SPLINE
SPL {X  -143.903, Y  +318.857, Z    +0.000, E1   +34.827, E3 +27306.081}
SPL {X  -153.845, Y  +344.850, Z    +0.000, E1   +24.318, E3 +27332.176}
SPL {X  -158.184, Y  +364.762, Z    +0.000, E1   +14.458, E3 +27341.556}
SPL {X  -159.644, Y  +378.137, Z    +0.000, E1    +6.763, E3 +27344.869}
SPL {X  -159.957, Y  +385.097, Z    +0.000, E1    +2.214, E3 +27345.786}
SPL {X  -160.000, Y  +390.467, Z    +0.000, E1    -1.886, E3 +27346.226}
SPL {X  -160.000, Y  +396.882, Z    +0.000, E1    -9.361, E3 +27346.979}
SPL {X  -160.000, Y  +403.298, Z    +0.000, E1   -17.340, E3 +27348.282}
SPL {X  -160.000, Y  +414.216, Z    +0.000, E1   -29.557, E3 +27351.832}
SPL {X  -160.000, Y  +448.199, Z    +0.000, E1   -47.246, E3 +27374.324}
SPL {X  -160.000, Y  +510.996, Z    +0.000, E1   -52.996, E3 +27446.648}
SPL {X  -160.000, Y  +527.680, Z    +0.000, E1   -53.008, E3 +27473.417}
SPL {X  -160.000, Y  +543.568, Z    +0.000, E1   -52.978, E3 +27498.957}
SPL {X  -160.000, Y  +558.178, Z    +0.000, E1   -52.971, E3 +27522.417}
SPL {X  -160.000, Y  +573.149, Z    +0.000, E1   -52.983, E3 +27546.431}
SPL {X  -160.000, Y  +589.074, Z    +0.000, E1   -52.998, E3 +27571.971}
SPL {X  -160.000, Y  +605.389, Z    +0.000, E1   -52.996, E3 +27598.171}
SPL {X  -160.000, Y  +621.194, Z    +0.000, E1   -52.986, E3 +27623.571}
SPL {X  -160.000, Y  +634.261, Z    +0.000, E1   -52.926, E3 +27644.650}
SPL {X  -160.000, Y  +645.165, Z    +0.000, E1   -52.917, E3 +27662.170}
SPL {X  -160.000, Y  +655.362, Z    +0.000, E1   -52.919, E3 +27678.521}
SPL {X  -160.000, Y  +666.642, Z    +0.000, E1   -52.938, E3 +27696.596}
SPL {X  -159.882, Y  +677.646, Z    +0.000, E1   -52.897, E3 +27714.427}
SPL {X  -159.100, Y  +688.445, Z    +0.000, E1   -52.790, E3 +27732.550}
SPL {X  -157.767, Y  +698.140, Z    +0.000, E1   -52.527, E3 +27749.561}
SPL {X  -155.944, Y  +707.296, Z    +0.000, E1   -52.232, E3 +27766.119}
SPL {X  -153.388, Y  +717.020, Z    +0.000, E1   -51.781, E3 +27784.324}
SPL {X  -150.628, Y  +725.455, Z    +0.000, E1   -51.252, E3 +27800.683}
SPL {X  -147.586, Y  +733.294, Z    +0.000, E1   -50.691, E3 +27816.259}
SPL {X  -144.002, Y  +741.239, Z    +0.000, E1   -50.009, E3 +27832.435}
SPL {X  -134.968, Y  +757.427, Z    +0.000, E1   -43.006, E3 +27917.714}
ENDSPLINE

SPLINE
SPL {X  -150.251, Y  +726.498, Z    +0.000, E1   -29.147, E3 +27992.699}
SPL {X  -158.295, Y  +694.796, Z    +0.000, E1   -14.337, E3 +28010.691}
SPL {X  -159.852, Y  +678.369, Z    +0.000, E1    -4.607, E3 +28014.636}
SPL {X  -159.994, Y  +672.856, Z    +0.000, E1    -0.741, E3 +28015.223}
SPL {X  -160.000, Y  +667.974, Z    +0.000, E1    +3.384, E3 +28015.651}
SPL {X  -160.000, Y  +657.936, Z    +0.000, E1   +15.171, E3 +28017.404}
SPL {X  -160.000, Y  +643.339, Z    +0.000, E1   +31.330, E3 +28022.395}
SPL {X  -160.000, Y  +606.884, Z    +0.000, E1   +47.933, E3 +28048.251}
SPL {X  -160.000, Y  +552.863, Z    +0.000, E1   +52.205, E3 +28114.055}
SPL {X  -160.000, Y  +541.250, Z    +0.000, E1   +52.128, E3 +28133.359}
SPL {X  -160.000, Y  +532.225, Z    +0.000, E1   +52.130, E3 +28148.267}
SPL {X  -160.000, Y  +522.908, Z    +0.000, E1   +52.129, E3 +28163.671}
SPL {X  -160.000, Y  +514.018, Z    +0.000, E1   +52.121, E3 +28178.355}
SPL {X  -160.000, Y  +502.148, Z    +0.000, E1   +52.197, E3 +28197.831}
SPL {X  -160.000, Y  +488.825, Z    +0.000, E1   +51.737, E3 +28222.876}
ENDSPLINE

SPLINE
SPL {X  -160.000, Y  +489.568, Z    +0.000, E1   +48.224, E3 +28241.900}
ENDSPLINE

SPLINE
SPL {X  -160.000, Y  +479.301, Z    +0.000, E1   +49.113, E3 +28255.778}
SPL {X  -160.000, Y  +468.407, Z    +0.000, E1   +50.011, E3 +28270.105}
SPL {X  -160.000, Y  +457.258, Z    +0.000, E1   +50.929, E3 +28284.090}
SPL {X  -160.000, Y  +444.555, Z    +0.000, E1   +51.931, E3 +28299.575}
SPL {X  -160.000, Y  +432.374, Z    +0.000, E1   +52.787, E3 +28314.199}
SPL {X  -160.000, Y  +422.570, Z    +0.000, E1   +53.120, E3 +28327.957}
SPL {X  -160.000, Y  +412.343, Z    +0.000, E1   +53.116, E3 +28344.264}
SPL {X  -160.000, Y  +402.505, Z    +0.000, E1   +53.115, E3 +28359.937}
SPL {X  -160.000, Y  +391.565, Z    +0.000, E1   +53.135, E3 +28377.344}
SPL {X  -159.782, Y  +380.451, Z    +0.000, E1   +53.086, E3 +28395.306}
SPL {X  -159.005, Y  +370.988, Z    +0.000, E1   +52.949, E3 +28411.205}
SPL {X  -157.765, Y  +362.152, Z    +0.000, E1   +52.730, E3 +28426.603}
SPL {X  -156.057, Y  +353.496, Z    +0.000, E1   +52.443, E3 +28442.142}
SPL {X  -153.530, Y  +343.760, Z    +0.000, E1   +52.025, E3 +28460.195}
SPL {X  -150.540, Y  +334.599, Z    +0.000, E1   +51.451, E3 +28477.843}
SPL {X  -147.202, Y  +326.099, Z    +0.000, E1   +50.843, E3 +28494.637}
SPL {X  -143.559, Y  +318.154, Z    +0.000, E1   +50.126, E3 +28510.784}
SPL {X  -132.920, Y  +299.736, Z    +0.000, E1   +44.141, E3 +28591.929}
ENDSPLINE

SPLINE
SPL {X  -143.903, Y  +318.857, Z    +0.000, E1   +34.827, E3 +28656.076}
SPL {X  -153.845, Y  +344.850, Z    +0.000, E1   +24.318, E3 +28682.171}
SPL {X  -158.184, Y  +364.762, Z    +0.000, E1   +14.458, E3 +28691.551}
SPL {X  -159.644, Y  +378.137, Z    +0.000, E1    +6.763, E3 +28694.864}
SPL {X  -159.957, Y  +385.097, Z    +0.000, E1    +2.214, E3 +28695.781}
SPL {X  -160.000, Y  +390.467, Z    +0.000, E1    -1.886, E3 +28696.222}
SPL {X  -160.000, Y  +396.882, Z    +0.000, E1    -9.361, E3 +28696.974}
SPL {X  -160.000, Y  +403.298, Z    +0.000, E1   -17.340, E3 +28698.277}
SPL {X  -160.000, Y  +414.216, Z    +0.000, E1   -29.557, E3 +28701.827}
SPL {X  -160.000, Y  +448.199, Z    +0.000, E1   -47.246, E3 +28724.319}
SPL {X  -160.000, Y  +510.996, Z    +0.000, E1   -52.996, E3 +28796.643}
SPL {X  -160.000, Y  +527.680, Z    +0.000, E1   -53.008, E3 +28823.412}
SPL {X  -160.000, Y  +543.568, Z    +0.000, E1   -52.978, E3 +28848.952}
SPL {X  -160.000, Y  +558.178, Z    +0.000, E1   -52.971, E3 +28872.412}
SPL {X  -160.000, Y  +573.149, Z    +0.000, E1   -52.983, E3 +28896.426}
SPL {X  -160.000, Y  +589.074, Z    +0.000, E1   -52.998, E3 +28921.966}
SPL {X  -160.000, Y  +605.389, Z    +0.000, E1   -52.996, E3 +28948.167}
SPL {X  -160.000, Y  +621.194, Z    +0.000, E1   -52.986, E3 +28973.566}
SPL {X  -160.000, Y  +634.261, Z    +0.000, E1   -52.926, E3 +28994.646}
SPL {X  -160.000, Y  +645.165, Z    +0.000, E1   -52.917, E3 +29012.165}
SPL {X  -160.000, Y  +655.362, Z    +0.000, E1   -52.919, E3 +29028.516}
SPL {X  -160.000, Y  +666.642, Z    +0.000, E1   -52.938, E3 +29046.591}
SPL {X  -159.882, Y  +677.646, Z    +0.000, E1   -52.897, E3 +29064.423}
SPL {X  -159.100, Y  +688.445, Z    +0.000, E1   -52.790, E3 +29082.545}
SPL {X  -157.767, Y  +698.140, Z    +0.000, E1   -52.527, E3 +29099.556}
SPL {X  -155.944, Y  +707.296, Z    +0.000, E1   -52.232, E3 +29116.115}
SPL {X  -153.388, Y  +717.020, Z    +0.000, E1   -51.781, E3 +29134.320}
SPL {X  -150.628, Y  +725.455, Z    +0.000, E1   -51.252, E3 +29150.678}
SPL {X  -147.586, Y  +733.294, Z    +0.000, E1   -50.691, E3 +29166.255}
SPL {X  -144.002, Y  +741.239, Z    +0.000, E1   -50.009, E3 +29182.431}
SPL {X  -134.968, Y  +757.427, Z    +0.000, E1   -43.006, E3 +29267.709}
ENDSPLINE

SPLINE
SPL {X  -150.251, Y  +726.498, Z    +0.000, E1   -29.147, E3 +29342.694}
SPL {X  -158.295, Y  +694.796, Z    +0.000, E1   -14.337, E3 +29360.687}
SPL {X  -159.852, Y  +678.369, Z    +0.000, E1    -4.607, E3 +29364.631}
SPL {X  -159.994, Y  +672.856, Z    +0.000, E1    -0.741, E3 +29365.219}
SPL {X  -160.000, Y  +667.974, Z    +0.000, E1    +3.384, E3 +29365.646}
SPL {X  -160.000, Y  +657.936, Z    +0.000, E1   +15.171, E3 +29367.399}
SPL {X  -160.000, Y  +643.339, Z    +0.000, E1   +31.330, E3 +29372.390}
SPL {X  -160.000, Y  +606.884, Z    +0.000, E1   +47.933, E3 +29398.246}
SPL {X  -160.000, Y  +552.863, Z    +0.000, E1   +52.205, E3 +29464.051}
SPL {X  -160.000, Y  +541.250, Z    +0.000, E1   +52.128, E3 +29483.354}
SPL {X  -160.000, Y  +532.225, Z    +0.000, E1   +52.130, E3 +29498.262}
SPL {X  -160.000, Y  +522.908, Z    +0.000, E1   +52.129, E3 +29513.666}
SPL {X  -160.000, Y  +514.018, Z    +0.000, E1   +52.121, E3 +29528.351}
SPL {X  -160.000, Y  +502.148, Z    +0.000, E1   +52.197, E3 +29547.827}
SPL {X  -160.000, Y  +488.825, Z    +0.000, E1   +51.737, E3 +29572.871}
ENDSPLINE

SPLINE
SPL {X  -160.000, Y  +489.568, Z    +0.000, E1   +48.224, E3 +29591.896}
ENDSPLINE

SPLINE
SPL {X  -160.000, Y  +479.301, Z    +0.000, E1   +49.113, E3 +29605.774}
SPL {X  -160.000, Y  +468.407, Z    +0.000, E1   +50.011, E3 +29620.100}
SPL {X  -160.000, Y  +457.258, Z    +0.000, E1   +50.929, E3 +29634.086}
SPL {X  -160.000, Y  +444.555, Z    +0.000, E1   +51.931, E3 +29649.570}
SPL {X  -160.000, Y  +432.374, Z    +0.000, E1   +52.787, E3 +29664.194}
SPL {X  -160.000, Y  +422.570, Z    +0.000, E1   +53.120, E3 +29677.952}
SPL {X  -160.000, Y  +412.343, Z    +0.000, E1   +53.116, E3 +29694.259}
SPL {X  -160.000, Y  +402.505, Z    +0.000, E1   +53.115, E3 +29709.932}
SPL {X  -160.000, Y  +391.565, Z    +0.000, E1   +53.135, E3 +29727.339}
SPL {X  -159.782, Y  +380.451, Z    +0.000, E1   +53.086, E3 +29745.301}
SPL {X  -159.005, Y  +370.988, Z    +0.000, E1   +52.949, E3 +29761.200}
SPL {X  -157.765, Y  +362.152, Z    +0.000, E1   +52.730, E3 +29776.599}
SPL {X  -156.057, Y  +353.496, Z    +0.000, E1   +52.443, E3 +29792.137}
SPL {X  -153.530, Y  +343.760, Z    +0.000, E1   +52.025, E3 +29810.190}
SPL {X  -150.540, Y  +334.599, Z    +0.000, E1   +51.451, E3 +29827.839}
SPL {X  -147.202, Y  +326.099, Z    +0.000, E1   +50.843, E3 +29844.632}
SPL {X  -143.559, Y  +318.154, Z    +0.000, E1   +50.126, E3 +29860.779}
SPL {X  -132.920, Y  +299.736, Z    +0.000, E1   +44.141, E3 +29941.924}
ENDSPLINE

SPLINE
SPL {X  -143.903, Y  +318.857, Z    +0.000, E1   +34.827, E3 +30006.071}
SPL {X  -153.845, Y  +344.850, Z    +0.000, E1   +24.318, E3 +30032.167}
SPL {X  -158.184, Y  +364.762, Z    +0.000, E1   +14.458, E3 +30041.546}
SPL {X  -159.644, Y  +378.137, Z    +0.000, E1    +6.763, E3 +30044.860}
SPL {X  -159.957, Y  +385.097, Z    +0.000, E1    +2.214, E3 +30045.776}
SPL {X  -160.000, Y  +390.467, Z    +0.000, E1    -1.886, E3 +30046.217}
SPL {X  -160.000, Y  +396.882, Z    +0.000, E1    -9.361, E3 +30046.970}
SPL {X  -160.000, Y  +403.298, Z    +0.000, E1   -17.340, E3 +30048.272}
SPL {X  -160.000, Y  +414.216, Z    +0.000, E1   -29.557, E3 +30051.822}
SPL {X  -160.000, Y  +448.199, Z    +0.000, E1   -47.246, E3 +30074.315}
SPL {X  -160.000, Y  +510.996, Z    +0.000, E1   -52.996, E3 +30146.639}
SPL {X  -160.000, Y  +527.680, Z    +0.000, E1   -53.008, E3 +30173.407}
SPL {X  -160.000, Y  +543.568, Z    +0.000, E1   -52.978, E3 +30198.947}
SPL {X  -160.000, Y  +558.178, Z    +0.000, E1   -52.971, E3 +30222.407}
SPL {X  -160.000, Y  +573.149, Z    +0.000, E1   -52.983, E3 +30246.421}
SPL {X  -160.000, Y  +589.074, Z    +0.000, E1   -52.998, E3 +30271.961}
SPL {X  -160.000, Y  +605.389, Z    +0.000, E1   -52.996, E3 +30298.162}
SPL {X  -160.000, Y  +621.194, Z    +0.000, E1   -52.986, E3 +30323.561}
SPL {X  -160.000, Y  +634.261, Z    +0.000, E1   -52.926, E3 +30344.641}
SPL {X  -160.000, Y  +645.165, Z    +0.000, E1   -52.917, E3 +30362.160}
SPL {X  -160.000, Y  +655.362, Z    +0.000, E1   -52.919, E3 +30378.511}
SPL {X  -160.000, Y  +666.642, Z    +0.000, E1   -52.938, E3 +30396.586}
SPL {X  -159.882, Y  +677.646, Z    +0.000, E1   -52.897, E3 +30414.418}
SPL {X  -159.100, Y  +688.445, Z    +0.000, E1   -52.790, E3 +30432.540}
SPL {X  -157.767, Y  +698.140, Z    +0.000, E1   -52.527, E3 +30449.552}
SPL {X  -155.944, Y  +707.296, Z    +0.000, E1   -52.232, E3 +30466.110}
SPL {X  -153.388, Y  +717.020, Z    +0.000, E1   -51.781, E3 +30484.315}
SPL {X  -150.628, Y  +725.455, Z    +0.000, E1   -51.252, E3 +30500.673}
SPL {X  -147.586, Y  +733.294, Z    +0.000, E1   -50.691, E3 +30516.250}
SPL {X  -144.002, Y  +741.239, Z    +0.000, E1   -50.009, E3 +30532.426}
SPL {X  -134.968, Y  +757.427, Z    +0.000, E1   -43.006, E3 +30617.704}
ENDSPLINE

SPLINE
SPL {X  -150.251, Y  +726.498, Z    +0.000, E1   -29.147, E3 +30692.690}
SPL {X  -158.295, Y  +694.796, Z    +0.000, E1   -14.337, E3 +30710.682}
SPL {X  -159.852, Y  +678.369, Z    +0.000, E1    -4.607, E3 +30714.626}
SPL {X  -159.994, Y  +672.856, Z    +0.000, E1    -0.741, E3 +30715.214}
SPL {X  -160.000, Y  +667.974, Z    +0.000, E1    +3.384, E3 +30715.642}
SPL {X  -160.000, Y  +657.936, Z    +0.000, E1   +15.171, E3 +30717.394}
SPL {X  -160.000, Y  +643.339, Z    +0.000, E1   +31.330, E3 +30722.386}
SPL {X  -160.000, Y  +606.884, Z    +0.000, E1   +47.933, E3 +30748.241}
SPL {X  -160.000, Y  +552.863, Z    +0.000, E1   +52.205, E3 +30814.046}
SPL {X  -160.000, Y  +541.250, Z    +0.000, E1   +52.128, E3 +30833.350}
SPL {X  -160.000, Y  +532.225, Z    +0.000, E1   +52.130, E3 +30848.257}
SPL {X  -160.000, Y  +522.908, Z    +0.000, E1   +52.129, E3 +30863.661}
SPL {X  -160.000, Y  +514.018, Z    +0.000, E1   +52.121, E3 +30878.346}
SPL {X  -160.000, Y  +502.148, Z    +0.000, E1   +52.197, E3 +30897.822}
SPL {X  -160.000, Y  +488.825, Z    +0.000, E1   +51.737, E3 +30922.867}
ENDSPLINE

SPLINE
SPL {X  -160.000, Y  +489.568, Z    +0.000, E1   +48.224, E3 +30941.891}
ENDSPLINE

SPLINE
SPL {X  -160.000, Y  +479.301, Z    +0.000, E1   +49.113, E3 +30955.769}
SPL {X  -160.000, Y  +468.407, Z    +0.000, E1   +50.011, E3 +30970.095}
SPL {X  -160.000, Y  +457.258, Z    +0.000, E1   +50.929, E3 +30984.081}
SPL {X  -160.000, Y  +444.555, Z    +0.000, E1   +51.931, E3 +30999.565}
SPL {X  -160.000, Y  +432.374, Z    +0.000, E1   +52.787, E3 +31014.189}
SPL {X  -160.000, Y  +422.570, Z    +0.000, E1   +53.120, E3 +31027.948}
SPL {X  -160.000, Y  +412.343, Z    +0.000, E1   +53.116, E3 +31044.254}
SPL {X  -160.000, Y  +402.505, Z    +0.000, E1   +53.115, E3 +31059.927}
SPL {X  -160.000, Y  +391.565, Z    +0.000, E1   +53.135, E3 +31077.334}
SPL {X  -159.782, Y  +380.451, Z    +0.000, E1   +53.086, E3 +31095.297}
SPL {X  -159.005, Y  +370.988, Z    +0.000, E1   +52.949, E3 +31111.195}
SPL {X  -157.765, Y  +362.152, Z    +0.000, E1   +52.730, E3 +31126.594}
SPL {X  -156.057, Y  +353.496, Z    +0.000, E1   +52.443, E3 +31142.132}
SPL {X  -153.530, Y  +343.760, Z    +0.000, E1   +52.025, E3 +31160.185}
SPL {X  -150.540, Y  +334.599, Z    +0.000, E1   +51.451, E3 +31177.834}
SPL {X  -147.202, Y  +326.099, Z    +0.000, E1   +50.843, E3 +31194.627}
SPL {X  -143.559, Y  +318.154, Z    +0.000, E1   +50.126, E3 +31210.775}
SPL {X  -132.920, Y  +299.736, Z    +0.000, E1   +44.141, E3 +31291.919}
ENDSPLINE

SPLINE
SPL {X  -143.903, Y  +318.857, Z    +0.000, E1   +34.827, E3 +31356.067}
SPL {X  -153.845, Y  +344.850, Z    +0.000, E1   +24.318, E3 +31382.162}
SPL {X  -158.184, Y  +364.762, Z    +0.000, E1   +14.458, E3 +31391.541}
SPL {X  -159.644, Y  +378.137, Z    +0.000, E1    +6.763, E3 +31394.855}
SPL {X  -159.957, Y  +385.097, Z    +0.000, E1    +2.214, E3 +31395.771}
SPL {X  -160.000, Y  +390.467, Z    +0.000, E1    -1.886, E3 +31396.212}
SPL {X  -160.000, Y  +396.882, Z    +0.000, E1    -9.361, E3 +31396.965}
SPL {X  -160.000, Y  +403.298, Z    +0.000, E1   -17.340, E3 +31398.268}
SPL {X  -160.000, Y  +414.216, Z    +0.000, E1   -29.557, E3 +31401.817}
SPL {X  -160.000, Y  +448.199, Z    +0.000, E1   -47.246, E3 +31424.310}
SPL {X  -160.000, Y  +510.996, Z    +0.000, E1   -52.996, E3 +31496.634}
SPL {X  -160.000, Y  +527.680, Z    +0.000, E1   -53.008, E3 +31523.403}
SPL {X  -160.000, Y  +543.568, Z    +0.000, E1   -52.978, E3 +31548.943}
SPL {X  -160.000, Y  +558.178, Z    +0.000, E1   -52.971, E3 +31572.402}
SPL {X  -160.000, Y  +573.149, Z    +0.000, E1   -52.983, E3 +31596.416}
SPL {X  -160.000, Y  +589.074, Z    +0.000, E1   -52.998, E3 +31621.957}
SPL {X  -160.000, Y  +605.389, Z    +0.000, E1   -52.996, E3 +31648.157}
SPL {X  -160.000, Y  +621.194, Z    +0.000, E1   -52.986, E3 +31673.557}
SPL {X  -160.000, Y  +634.261, Z    +0.000, E1   -52.926, E3 +31694.636}
SPL {X  -160.000, Y  +645.165, Z    +0.000, E1   -52.917, E3 +31712.155}
SPL {X  -160.000, Y  +655.362, Z    +0.000, E1   -52.919, E3 +31728.506}
SPL {X  -160.000, Y  +666.642, Z    +0.000, E1   -52.938, E3 +31746.582}
SPL {X  -159.882, Y  +677.646, Z    +0.000, E1   -52.897, E3 +31764.413}
SPL {X  -159.100, Y  +688.445, Z    +0.000, E1   -52.790, E3 +31782.536}
SPL {X  -157.767, Y  +698.140, Z    +0.000, E1   -52.527, E3 +31799.547}
SPL {X  -155.944, Y  +707.296, Z    +0.000, E1   -52.232, E3 +31816.105}
SPL {X  -153.388, Y  +717.020, Z    +0.000, E1   -51.781, E3 +31834.310}
SPL {X  -150.628, Y  +725.455, Z    +0.000, E1   -51.252, E3 +31850.668}
SPL {X  -147.586, Y  +733.294, Z    +0.000, E1   -50.691, E3 +31866.245}
SPL {X  -144.002, Y  +741.239, Z    +0.000, E1   -50.009, E3 +31882.421}
SPL {X  -134.968, Y  +757.427, Z    +0.000, E1   -43.006, E3 +31967.700}
ENDSPLINE

SPLINE
SPL {X  -150.251, Y  +726.498, Z    +0.000, E1   -29.147, E3 +32042.685}
SPL {X  -158.295, Y  +694.796, Z    +0.000, E1   -14.337, E3 +32060.677}
SPL {X  -159.852, Y  +678.369, Z    +0.000, E1    -4.607, E3 +32064.621}
SPL {X  -159.994, Y  +672.856, Z    +0.000, E1    -0.741, E3 +32065.209}
SPL {X  -160.000, Y  +667.974, Z    +0.000, E1    +3.384, E3 +32065.637}
SPL {X  -160.000, Y  +657.936, Z    +0.000, E1   +15.171, E3 +32067.389}
SPL {X  -160.000, Y  +643.339, Z    +0.000, E1   +31.330, E3 +32072.381}
SPL {X  -160.000, Y  +606.884, Z    +0.000, E1   +47.933, E3 +32098.236}
SPL {X  -160.000, Y  +552.863, Z    +0.000, E1   +52.205, E3 +32164.041}
SPL {X  -160.000, Y  +541.250, Z    +0.000, E1   +52.128, E3 +32183.345}
SPL {X  -160.000, Y  +532.225, Z    +0.000, E1   +52.130, E3 +32198.253}
SPL {X  -160.000, Y  +522.908, Z    +0.000, E1   +52.129, E3 +32213.656}
SPL {X  -160.000, Y  +514.018, Z    +0.000, E1   +52.121, E3 +32228.341}
SPL {X  -160.000, Y  +502.148, Z    +0.000, E1   +52.197, E3 +32247.817}
SPL {X  -160.000, Y  +488.825, Z    +0.000, E1   +51.737, E3 +32272.862}
ENDSPLINE

SPLINE
SPL {X  -160.000, Y  +489.568, Z    +0.000, E1   +48.224, E3 +32291.886}
ENDSPLINE

SPLINE
SPL {X  -160.000, Y  +479.301, Z    +0.000, E1   +49.113, E3 +32305.764}
SPL {X  -160.000, Y  +468.407, Z    +0.000, E1   +50.011, E3 +32320.091}
SPL {X  -160.000, Y  +457.258, Z    +0.000, E1   +50.929, E3 +32334.076}
SPL {X  -160.000, Y  +444.555, Z    +0.000, E1   +51.931, E3 +32349.560}
SPL {X  -160.000, Y  +432.374, Z    +0.000, E1   +52.787, E3 +32364.185}
SPL {X  -160.000, Y  +422.570, Z    +0.000, E1   +53.120, E3 +32377.943}
SPL {X  -160.000, Y  +412.343, Z    +0.000, E1   +53.116, E3 +32394.250}
SPL {X  -160.000, Y  +402.505, Z    +0.000, E1   +53.115, E3 +32409.923}
SPL {X  -160.000, Y  +391.565, Z    +0.000, E1   +53.135, E3 +32427.329}
SPL {X  -159.782, Y  +380.451, Z    +0.000, E1   +53.086, E3 +32445.292}
SPL {X  -159.005, Y  +370.988, Z    +0.000, E1   +52.949, E3 +32461.191}
SPL {X  -157.765, Y  +362.152, Z    +0.000, E1   +52.730, E3 +32476.589}
SPL {X  -156.057, Y  +353.496, Z    +0.000, E1   +52.443, E3 +32492.128}
SPL {X  -153.530, Y  +343.760, Z    +0.000, E1   +52.025, E3 +32510.181}
SPL {X  -150.540, Y  +334.599, Z    +0.000, E1   +51.451, E3 +32527.829}
SPL {X  -147.202, Y  +326.099, Z    +0.000, E1   +50.843, E3 +32544.623}
SPL {X  -143.559, Y  +318.154, Z    +0.000, E1   +50.126, E3 +32560.770}
SPL {X  -132.920, Y  +299.736, Z    +0.000, E1   +44.141, E3 +32641.914}
ENDSPLINE

SPLINE
SPL {X  -143.903, Y  +318.857, Z    +0.000, E1   +34.827, E3 +32706.062}
SPL {X  -153.845, Y  +344.850, Z    +0.000, E1   +24.318, E3 +32732.157}
SPL {X  -158.184, Y  +364.762, Z    +0.000, E1   +14.458, E3 +32741.537}
SPL {X  -159.644, Y  +378.137, Z    +0.000, E1    +6.763, E3 +32744.850}
SPL {X  -159.957, Y  +385.097, Z    +0.000, E1    +2.214, E3 +32745.767}
SPL {X  -160.000, Y  +390.467, Z    +0.000, E1    -1.886, E3 +32746.207}
SPL {X  -160.000, Y  +396.882, Z    +0.000, E1    -9.361, E3 +32746.960}
SPL {X  -160.000, Y  +403.298, Z    +0.000, E1   -17.340, E3 +32748.263}
SPL {X  -160.000, Y  +414.216, Z    +0.000, E1   -29.557, E3 +32751.813}
SPL {X  -160.000, Y  +448.199, Z    +0.000, E1   -47.246, E3 +32774.305}
SPL {X  -160.000, Y  +510.996, Z    +0.000, E1   -52.996, E3 +32846.629}
SPL {X  -160.000, Y  +527.680, Z    +0.000, E1   -53.008, E3 +32873.398}
SPL {X  -160.000, Y  +543.568, Z    +0.000, E1   -52.978, E3 +32898.938}
SPL {X  -160.000, Y  +558.178, Z    +0.000, E1   -52.971, E3 +32922.398}
SPL {X  -160.000, Y  +573.149, Z    +0.000, E1   -52.983, E3 +32946.412}
SPL {X  -160.000, Y  +589.074, Z    +0.000, E1   -52.998, E3 +32971.952}
SPL {X  -160.000, Y  +605.389, Z    +0.000, E1   -52.996, E3 +32998.152}
SPL {X  -160.000, Y  +621.194, Z    +0.000, E1   -52.986, E3 +33023.552}
SPL {X  -160.000, Y  +634.261, Z    +0.000, E1   -52.926, E3 +33044.632}
SPL {X  -160.000, Y  +645.165, Z    +0.000, E1   -52.917, E3 +33062.151}
SPL {X  -160.000, Y  +655.362, Z    +0.000, E1   -52.919, E3 +33078.502}
SPL {X  -160.000, Y  +666.642, Z    +0.000, E1   -52.938, E3 +33096.577}
SPL {X  -159.882, Y  +677.646, Z    +0.000, E1   -52.897, E3 +33114.409}
SPL {X  -159.100, Y  +688.445, Z    +0.000, E1   -52.790, E3 +33132.531}
SPL {X  -157.767, Y  +698.140, Z    +0.000, E1   -52.527, E3 +33149.542}
SPL {X  -155.944, Y  +707.296, Z    +0.000, E1   -52.232, E3 +33166.100}
SPL {X  -153.388, Y  +717.020, Z    +0.000, E1   -51.781, E3 +33184.305}
SPL {X  -150.628, Y  +725.455, Z    +0.000, E1   -51.252, E3 +33200.664}
SPL {X  -147.586, Y  +733.294, Z    +0.000, E1   -50.691, E3 +33216.240}
SPL {X  -144.002, Y  +741.239, Z    +0.000, E1   -50.009, E3 +33232.417}
SPL {X  -134.968, Y  +757.427, Z    +0.000, E1   -43.006, E3 +33317.695}
ENDSPLINE

SPLINE
SPL {X  -150.251, Y  +726.498, Z    +0.000, E1   -29.147, E3 +33392.680}
SPL {X  -158.295, Y  +694.796, Z    +0.000, E1   -14.337, E3 +33410.672}
SPL {X  -159.852, Y  +678.369, Z    +0.000, E1    -4.607, E3 +33414.617}
SPL {X  -159.994, Y  +672.856, Z    +0.000, E1    -0.741, E3 +33415.204}
SPL {X  -160.000, Y  +667.974, Z    +0.000, E1    +3.384, E3 +33415.632}
SPL {X  -160.000, Y  +657.936, Z    +0.000, E1   +15.171, E3 +33417.385}
SPL {X  -160.000, Y  +643.339, Z    +0.000, E1   +31.330, E3 +33422.376}
SPL {X  -160.000, Y  +606.884, Z    +0.000, E1   +47.933, E3 +33448.232}
SPL {X  -160.000, Y  +552.863, Z    +0.000, E1   +52.205, E3 +33514.036}
SPL {X  -160.000, Y  +541.250, Z    +0.000, E1   +52.128, E3 +33533.340}
SPL {X  -160.000, Y  +532.225, Z    +0.000, E1   +52.130, E3 +33548.248}
SPL {X  -160.000, Y  +522.908, Z    +0.000, E1   +52.129, E3 +33563.652}
SPL {X  -160.000, Y  +514.018, Z    +0.000, E1   +52.121, E3 +33578.336}
SPL {X  -160.000, Y  +502.148, Z    +0.000, E1   +52.197, E3 +33597.812}
SPL {X  -160.000, Y  +488.825, Z    +0.000, E1   +51.737, E3 +33622.857}
ENDSPLINE

SPLINE
SPL {X  -160.000, Y  +489.568, Z    +0.000, E1   +48.224, E3 +33641.881}
ENDSPLINE

SPLINE
SPL {X  -160.000, Y  +479.301, Z    +0.000, E1   +49.113, E3 +33655.759}
SPL {X  -160.000, Y  +468.407, Z    +0.000, E1   +50.011, E3 +33670.086}
SPL {X  -160.000, Y  +457.258, Z    +0.000, E1   +50.929, E3 +33684.071}
SPL {X  -160.000, Y  +444.555, Z    +0.000, E1   +51.931, E3 +33699.556}
SPL {X  -160.000, Y  +432.374, Z    +0.000, E1   +52.787, E3 +33714.180}
SPL {X  -160.000, Y  +422.570, Z    +0.000, E1   +53.120, E3 +33727.938}
SPL {X  -160.000, Y  +412.343, Z    +0.000, E1   +53.116, E3 +33744.245}
SPL {X  -160.000, Y  +402.505, Z    +0.000, E1   +53.115, E3 +33759.918}
SPL {X  -160.000, Y  +391.565, Z    +0.000, E1   +53.135, E3 +33777.325}
SPL {X  -159.782, Y  +380.451, Z    +0.000, E1   +53.086, E3 +33795.287}
SPL {X  -159.005, Y  +370.988, Z    +0.000, E1   +52.949, E3 +33811.186}
SPL {X  -157.765, Y  +362.152, Z    +0.000, E1   +52.730, E3 +33826.584}
SPL {X  -156.057, Y  +353.496, Z    +0.000, E1   +52.443, E3 +33842.123}
SPL {X  -153.530, Y  +343.760, Z    +0.000, E1   +52.025, E3 +33860.176}
SPL {X  -150.540, Y  +334.599, Z    +0.000, E1   +51.451, E3 +33877.824}
SPL {X  -147.202, Y  +326.099, Z    +0.000, E1   +50.843, E3 +33894.618}
SPL {X  -143.559, Y  +318.154, Z    +0.000, E1   +50.126, E3 +33910.765}
SPL {X  -132.920, Y  +299.736, Z    +0.000, E1   +44.141, E3 +33991.910}
ENDSPLINE

SPLINE
SPL {X  -143.903, Y  +318.857, Z    +0.000, E1   +34.827, E3 +34056.057}
SPL {X  -153.845, Y  +344.850, Z    +0.000, E1   +24.318, E3 +34082.152}
SPL {X  -158.184, Y  +364.762, Z    +0.000, E1   +14.458, E3 +34091.532}
SPL {X  -159.644, Y  +378.137, Z    +0.000, E1    +6.763, E3 +34094.845}
SPL {X  -159.957, Y  +385.097, Z    +0.000, E1    +2.214, E3 +34095.762}
SPL {X  -160.000, Y  +390.467, Z    +0.000, E1    -1.886, E3 +34096.203}
SPL {X  -160.000, Y  +396.882, Z    +0.000, E1    -9.361, E3 +34096.955}
SPL {X  -160.000, Y  +403.298, Z    +0.000, E1   -17.340, E3 +34098.258}
SPL {X  -160.000, Y  +414.216, Z    +0.000, E1   -29.557, E3 +34101.808}
SPL {X  -160.000, Y  +448.199, Z    +0.000, E1   -47.246, E3 +34124.301}
SPL {X  -160.000, Y  +510.996, Z    +0.000, E1   -52.996, E3 +34196.624}
SPL {X  -160.000, Y  +527.680, Z    +0.000, E1   -53.008, E3 +34223.393}
SPL {X  -160.000, Y  +543.568, Z    +0.000, E1   -52.978, E3 +34248.933}
SPL {X  -160.000, Y  +558.178, Z    +0.000, E1   -52.971, E3 +34272.393}
SPL {X  -160.000, Y  +573.149, Z    +0.000, E1   -52.983, E3 +34296.407}
SPL {X  -160.000, Y  +589.074, Z    +0.000, E1   -52.998, E3 +34321.947}
SPL {X  -160.000, Y  +605.389, Z    +0.000, E1   -52.996, E3 +34348.148}
SPL {X  -160.000, Y  +621.194, Z    +0.000, E1   -52.986, E3 +34373.547}
SPL {X  -160.000, Y  +634.261, Z    +0.000, E1   -52.926, E3 +34394.627}
SPL {X  -160.000, Y  +645.165, Z    +0.000, E1   -52.917, E3 +34412.146}
SPL {X  -160.000, Y  +655.362, Z    +0.000, E1   -52.919, E3 +34428.497}
SPL {X  -160.000, Y  +666.642, Z    +0.000, E1   -52.938, E3 +34446.572}
SPL {X  -159.882, Y  +677.646, Z    +0.000, E1   -52.897, E3 +34464.404}
SPL {X  -159.100, Y  +688.445, Z    +0.000, E1   -52.790, E3 +34482.526}
SPL {X  -157.767, Y  +698.140, Z    +0.000, E1   -52.527, E3 +34499.537}
SPL {X  -155.944, Y  +707.296, Z    +0.000, E1   -52.232, E3 +34516.096}
SPL {X  -153.388, Y  +717.020, Z    +0.000, E1   -51.781, E3 +34534.301}
SPL {X  -150.628, Y  +725.455, Z    +0.000, E1   -51.252, E3 +34550.659}
SPL {X  -147.586, Y  +733.294, Z    +0.000, E1   -50.691, E3 +34566.236}
SPL {X  -144.002, Y  +741.239, Z    +0.000, E1   -50.009, E3 +34582.412}
SPL {X  -134.968, Y  +757.427, Z    +0.000, E1   -43.006, E3 +34667.690}
ENDSPLINE

SPLINE
SPL {X  -150.251, Y  +726.498, Z    +0.000, E1   -29.147, E3 +34742.675}
SPL {X  -158.295, Y  +694.796, Z    +0.000, E1   -14.337, E3 +34760.668}
SPL {X  -159.852, Y  +678.369, Z    +0.000, E1    -4.607, E3 +34764.612}
SPL {X  -159.994, Y  +672.856, Z    +0.000, E1    -0.741, E3 +34765.200}
SPL {X  -160.000, Y  +667.974, Z    +0.000, E1    +3.384, E3 +34765.627}
SPL {X  -160.000, Y  +657.936, Z    +0.000, E1   +15.171, E3 +34767.380}
SPL {X  -160.000, Y  +643.339, Z    +0.000, E1   +31.330, E3 +34772.372}
SPL {X  -160.000, Y  +606.884, Z    +0.000, E1   +47.933, E3 +34798.227}
SPL {X  -160.000, Y  +552.863, Z    +0.000, E1   +52.205, E3 +34864.032}
SPL {X  -160.000, Y  +541.250, Z    +0.000, E1   +52.128, E3 +34883.336}
SPL {X  -160.000, Y  +532.225, Z    +0.000, E1   +52.130, E3 +34898.243}
SPL {X  -160.000, Y  +522.908, Z    +0.000, E1   +52.129, E3 +34913.647}
SPL {X  -160.000, Y  +514.018, Z    +0.000, E1   +52.121, E3 +34928.332}
SPL {X  -160.000, Y  +502.148, Z    +0.000, E1   +52.197, E3 +34947.808}
SPL {X  -160.000, Y  +488.825, Z    +0.000, E1   +51.737, E3 +34972.852}
ENDSPLINE

SPLINE
SPL {X  -160.000, Y  +489.568, Z    +0.000, E1   +48.224, E3 +34991.877}
ENDSPLINE

SPLINE
SPL {X  -160.000, Y  +479.301, Z    +0.000, E1   +49.113, E3 +35005.755}
SPL {X  -160.000, Y  +468.407, Z    +0.000, E1   +50.011, E3 +35020.081}
SPL {X  -160.000, Y  +457.258, Z    +0.000, E1   +50.929, E3 +35034.067}
SPL {X  -160.000, Y  +444.555, Z    +0.000, E1   +51.931, E3 +35049.551}
SPL {X  -160.000, Y  +432.374, Z    +0.000, E1   +52.787, E3 +35064.175}
SPL {X  -160.000, Y  +422.570, Z    +0.000, E1   +53.120, E3 +35077.933}
SPL {X  -160.000, Y  +412.343, Z    +0.000, E1   +53.116, E3 +35094.240}
SPL {X  -160.000, Y  +402.505, Z    +0.000, E1   +53.115, E3 +35109.913}
SPL {X  -160.000, Y  +391.565, Z    +0.000, E1   +53.135, E3 +35127.320}
SPL {X  -159.782, Y  +380.451, Z    +0.000, E1   +53.086, E3 +35145.282}
SPL {X  -159.005, Y  +370.988, Z    +0.000, E1   +52.949, E3 +35161.181}
SPL {X  -157.765, Y  +362.152, Z    +0.000, E1   +52.730, E3 +35176.580}
SPL {X  -156.057, Y  +353.496, Z    +0.000, E1   +52.443, E3 +35192.118}
SPL {X  -153.530, Y  +343.760, Z    +0.000, E1   +52.025, E3 +35210.171}
SPL {X  -150.540, Y  +334.599, Z    +0.000, E1   +51.451, E3 +35227.820}
SPL {X  -147.202, Y  +326.099, Z    +0.000, E1   +50.843, E3 +35244.613}
SPL {X  -143.559, Y  +318.154, Z    +0.000, E1   +50.126, E3 +35260.760}
SPL {X  -132.920, Y  +299.736, Z    +0.000, E1   +44.141, E3 +35341.905}
ENDSPLINE

SPLINE
SPL {X  -143.903, Y  +318.857, Z    +0.000, E1   +34.827, E3 +35406.052}
SPL {X  -153.845, Y  +344.850, Z    +0.000, E1   +24.318, E3 +35432.148}
SPL {X  -158.184, Y  +364.762, Z    +0.000, E1   +14.458, E3 +35441.527}
SPL {X  -159.644, Y  +378.137, Z    +0.000, E1    +6.763, E3 +35444.841}
SPL {X  -159.957, Y  +385.097, Z    +0.000, E1    +2.214, E3 +35445.757}
SPL {X  -160.000, Y  +390.467, Z    +0.000, E1    -1.886, E3 +35446.198}
SPL {X  -160.000, Y  +396.882, Z    +0.000, E1    -9.361, E3 +35446.951}
SPL {X  -160.000, Y  +403.298, Z    +0.000, E1   -17.340, E3 +35448.253}
SPL {X  -160.000, Y  +414.216, Z    +0.000, E1   -29.557, E3 +35451.803}
SPL {X  -160.000, Y  +448.199, Z    +0.000, E1   -47.246, E3 +35474.296}
SPL {X  -160.000, Y  +510.996, Z    +0.000, E1   -52.996, E3 +35546.620}
SPL {X  -160.000, Y  +527.680, Z    +0.000, E1   -53.008, E3 +35573.388}
SPL {X  -160.000, Y  +543.568, Z    +0.000, E1   -52.978, E3 +35598.928}
SPL {X  -160.000, Y  +558.178, Z    +0.000, E1   -52.971, E3 +35622.388}
SPL {X  -160.000, Y  +573.149, Z    +0.000, E1   -52.983, E3 +35646.402}
SPL {X  -160.000, Y  +589.074, Z    +0.000, E1   -52.998, E3 +35671.942}
SPL {X  -160.000, Y  +605.389, Z    +0.000, E1   -52.996, E3 +35698.143}
SPL {X  -160.000, Y  +621.194, Z    +0.000, E1   -52.986, E3 +35723.542}
SPL {X  -160.000, Y  +634.261, Z    +0.000, E1   -52.926, E3 +35744.622}
SPL {X  -160.000, Y  +645.165, Z    +0.000, E1   -52.917, E3 +35762.141}
SPL {X  -160.000, Y  +655.362, Z    +0.000, E1   -52.919, E3 +35778.492}
SPL {X  -160.000, Y  +666.642, Z    +0.000, E1   -52.938, E3 +35796.567}
SPL {X  -159.882, Y  +677.646, Z    +0.000, E1   -52.897, E3 +35814.399}
SPL {X  -159.100, Y  +688.445, Z    +0.000, E1   -52.790, E3 +35832.521}
SPL {X  -157.767, Y  +698.140, Z    +0.000, E1   -52.527, E3 +35849.533}
SPL {X  -155.944, Y  +707.296, Z    +0.000, E1   -52.232, E3 +35866.091}
SPL {X  -153.388, Y  +717.020, Z    +0.000, E1   -51.781, E3 +35884.296}
SPL {X  -150.628, Y  +725.455, Z    +0.000, E1   -51.252, E3 +35900.654}
SPL {X  -147.586, Y  +733.294, Z    +0.000, E1   -50.691, E3 +35916.231}
SPL {X  -144.002, Y  +741.239, Z    +0.000, E1   -50.009, E3 +35932.407}
SPL {X  -134.968, Y  +757.427, Z    +0.000, E1   -43.006, E3 +36017.685}
ENDSPLINE

SPLINE
SPL {X  -150.251, Y  +726.498, Z    +0.000, E1   -29.147, E3 +36092.671}
SPL {X  -158.295, Y  +694.796, Z    +0.000, E1   -14.337, E3 +36110.663}
SPL {X  -159.852, Y  +678.369, Z    +0.000, E1    -4.607, E3 +36114.607}
SPL {X  -159.994, Y  +672.856, Z    +0.000, E1    -0.741, E3 +36115.195}
SPL {X  -160.000, Y  +667.974, Z    +0.000, E1    +3.384, E3 +36115.623}
SPL {X  -160.000, Y  +657.936, Z    +0.000, E1   +15.171, E3 +36117.375}
SPL {X  -160.000, Y  +643.339, Z    +0.000, E1   +31.330, E3 +36122.367}
SPL {X  -160.000, Y  +606.884, Z    +0.000, E1   +47.933, E3 +36148.222}
SPL {X  -160.000, Y  +552.863, Z    +0.000, E1   +52.205, E3 +36214.027}
SPL {X  -160.000, Y  +541.250, Z    +0.000, E1   +52.128, E3 +36233.331}
SPL {X  -160.000, Y  +532.225, Z    +0.000, E1   +52.130, E3 +36248.238}
SPL {X  -160.000, Y  +522.908, Z    +0.000, E1   +52.129, E3 +36263.642}
SPL {X  -160.000, Y  +514.018, Z    +0.000, E1   +52.121, E3 +36278.327}
SPL {X  -160.000, Y  +502.148, Z    +0.000, E1   +52.197, E3 +36297.803}
SPL {X  -160.000, Y  +488.825, Z    +0.000, E1   +51.737, E3 +36322.848}
ENDSPLINE

SPLINE
SPL {X  -160.000, Y  +489.568, Z    +0.000, E1   +48.224, E3 +36341.872}
ENDSPLINE

SPLINE
SPL {X  -160.000, Y  +479.301, Z    +0.000, E1   +49.113, E3 +36355.750}
SPL {X  -160.000, Y  +468.407, Z    +0.000, E1   +50.011, E3 +36370.076}
SPL {X  -160.000, Y  +457.258, Z    +0.000, E1   +50.929, E3 +36384.062}
SPL {X  -160.000, Y  +444.555, Z    +0.000, E1   +51.931, E3 +36399.546}
SPL {X  -160.000, Y  +432.374, Z    +0.000, E1   +52.787, E3 +36414.170}
SPL {X  -160.000, Y  +422.570, Z    +0.000, E1   +53.120, E3 +36427.929}
SPL {X  -160.000, Y  +412.343, Z    +0.000, E1   +53.116, E3 +36444.235}
SPL {X  -160.000, Y  +402.505, Z    +0.000, E1   +53.115, E3 +36459.908}
SPL {X  -160.000, Y  +391.565, Z    +0.000, E1   +53.135, E3 +36477.315}
SPL {X  -159.782, Y  +380.451, Z    +0.000, E1   +53.086, E3 +36495.278}
SPL {X  -159.005, Y  +370.988, Z    +0.000, E1   +52.949, E3 +36511.176}
SPL {X  -157.765, Y  +362.152, Z    +0.000, E1   +52.730, E3 +36526.575}
SPL {X  -156.057, Y  +353.496, Z    +0.000, E1   +52.443, E3 +36542.113}
SPL {X  -153.530, Y  +343.760, Z    +0.000, E1   +52.025, E3 +36560.166}
SPL {X  -150.540, Y  +334.599, Z    +0.000, E1   +51.451, E3 +36577.815}
SPL {X  -147.202, Y  +326.099, Z    +0.000, E1   +50.843, E3 +36594.608}
SPL {X  -143.559, Y  +318.154, Z    +0.000, E1   +50.126, E3 +36610.756}
SPL {X  -132.920, Y  +299.736, Z    +0.000, E1   +44.141, E3 +36691.900}
ENDSPLINE

SPLINE
SPL {X  -143.903, Y  +318.857, Z    +0.000, E1   +34.827, E3 +36756.048}
SPL {X  -153.845, Y  +344.850, Z    +0.000, E1   +24.318, E3 +36782.143}
SPL {X  -158.184, Y  +364.762, Z    +0.000, E1   +14.458, E3 +36791.522}
SPL {X  -159.644, Y  +378.137, Z    +0.000, E1    +6.763, E3 +36794.836}
SPL {X  -159.957, Y  +385.097, Z    +0.000, E1    +2.214, E3 +36795.753}
SPL {X  -160.000, Y  +390.467, Z    +0.000, E1    -1.886, E3 +36796.193}
SPL {X  -160.000, Y  +396.882, Z    +0.000, E1    -9.361, E3 +36796.946}
SPL {X  -160.000, Y  +403.298, Z    +0.000, E1   -17.340, E3 +36798.249}
SPL {X  -160.000, Y  +414.216, Z    +0.000, E1   -29.557, E3 +36801.798}
SPL {X  -160.000, Y  +448.199, Z    +0.000, E1   -47.246, E3 +36824.291}
SPL {X  -160.000, Y  +510.996, Z    +0.000, E1   -52.996, E3 +36896.615}
SPL {X  -160.000, Y  +527.680, Z    +0.000, E1   -53.008, E3 +36923.384}
SPL {X  -160.000, Y  +543.568, Z    +0.000, E1   -52.978, E3 +36948.924}
SPL {X  -160.000, Y  +558.178, Z    +0.000, E1   -52.971, E3 +36972.383}
SPL {X  -160.000, Y  +573.149, Z    +0.000, E1   -52.983, E3 +36996.397}
SPL {X  -160.000, Y  +589.074, Z    +0.000, E1   -52.998, E3 +37021.938}
SPL {X  -160.000, Y  +605.389, Z    +0.000, E1   -52.996, E3 +37048.138}
SPL {X  -160.000, Y  +621.194, Z    +0.000, E1   -52.986, E3 +37073.538}
SPL {X  -160.000, Y  +634.261, Z    +0.000, E1   -52.926, E3 +37094.617}
SPL {X  -160.000, Y  +645.165, Z    +0.000, E1   -52.917, E3 +37112.136}
SPL {X  -160.000, Y  +655.362, Z    +0.000, E1   -52.919, E3 +37128.488}
SPL {X  -160.000, Y  +666.642, Z    +0.000, E1   -52.938, E3 +37146.563}
SPL {X  -159.882, Y  +677.646, Z    +0.000, E1   -52.897, E3 +37164.394}
SPL {X  -159.100, Y  +688.445, Z    +0.000, E1   -52.790, E3 +37182.517}
SPL {X  -157.767, Y  +698.140, Z    +0.000, E1   -52.527, E3 +37199.528}
SPL {X  -155.944, Y  +707.296, Z    +0.000, E1   -52.232, E3 +37216.086}
SPL {X  -153.388, Y  +717.020, Z    +0.000, E1   -51.781, E3 +37234.291}
SPL {X  -150.628, Y  +725.455, Z    +0.000, E1   -51.252, E3 +37250.649}
SPL {X  -147.586, Y  +733.294, Z    +0.000, E1   -50.691, E3 +37266.226}
SPL {X  -144.002, Y  +741.239, Z    +0.000, E1   -50.009, E3 +37282.402}
SPL {X  -134.968, Y  +757.427, Z    +0.000, E1   -43.006, E3 +37367.681}
ENDSPLINE

SPLINE
SPL {X  -150.251, Y  +726.498, Z    +0.000, E1   -29.147, E3 +37442.666}
SPL {X  -158.295, Y  +694.796, Z    +0.000, E1   -14.337, E3 +37460.658}
SPL {X  -159.852, Y  +678.369, Z    +0.000, E1    -4.607, E3 +37464.602}
SPL {X  -159.994, Y  +672.856, Z    +0.000, E1    -0.741, E3 +37465.190}
SPL {X  -160.000, Y  +667.974, Z    +0.000, E1    +3.384, E3 +37465.618}
SPL {X  -160.000, Y  +657.936, Z    +0.000, E1   +15.171, E3 +37467.370}
SPL {X  -160.000, Y  +643.339, Z    +0.000, E1   +31.330, E3 +37472.362}
SPL {X  -160.000, Y  +606.884, Z    +0.000, E1   +47.933, E3 +37498.217}
SPL {X  -160.000, Y  +552.863, Z    +0.000, E1   +52.205, E3 +37564.022}
SPL {X  -160.000, Y  +541.250, Z    +0.000, E1   +52.128, E3 +37583.326}
SPL {X  -160.000, Y  +532.225, Z    +0.000, E1   +52.130, E3 +37598.234}
SPL {X  -160.000, Y  +522.908, Z    +0.000, E1   +52.129, E3 +37613.637}
SPL {X  -160.000, Y  +514.018, Z    +0.000, E1   +52.121, E3 +37628.322}
SPL {X  -160.000, Y  +502.148, Z    +0.000, E1   +52.197, E3 +37647.798}
SPL {X  -160.000, Y  +488.825, Z    +0.000, E1   +51.737, E3 +37672.843}
ENDSPLINE

SPLINE
SPL {X  -160.000, Y  +489.568, Z    +0.000, E1   +48.224, E3 +37691.867}
ENDSPLINE

SPLINE
SPL {X  -160.000, Y  +479.301, Z    +0.000, E1   +49.113, E3 +37705.745}
SPL {X  -160.000, Y  +468.407, Z    +0.000, E1   +50.011, E3 +37720.072}
SPL {X  -160.000, Y  +457.258, Z    +0.000, E1   +50.929, E3 +37734.057}
SPL {X  -160.000, Y  +444.555, Z    +0.000, E1   +51.931, E3 +37749.541}
SPL {X  -160.000, Y  +432.374, Z    +0.000, E1   +52.787, E3 +37764.166}
SPL {X  -160.000, Y  +422.570, Z    +0.000, E1   +53.120, E3 +37777.924}
SPL {X  -160.000, Y  +412.343, Z    +0.000, E1   +53.116, E3 +37794.231}
SPL {X  -160.000, Y  +402.505, Z    +0.000, E1   +53.115, E3 +37809.904}
SPL {X  -160.000, Y  +391.565, Z    +0.000, E1   +53.135, E3 +37827.310}
SPL {X  -159.782, Y  +380.451, Z    +0.000, E1   +53.086, E3 +37845.273}
SPL {X  -159.005, Y  +370.988, Z    +0.000, E1   +52.949, E3 +37861.172}
SPL {X  -157.765, Y  +362.152, Z    +0.000, E1   +52.730, E3 +37876.570}
SPL {X  -156.057, Y  +353.496, Z    +0.000, E1   +52.443, E3 +37892.109}
SPL {X  -153.530, Y  +343.760, Z    +0.000, E1   +52.025, E3 +37910.162}
SPL {X  -150.540, Y  +334.599, Z    +0.000, E1   +51.451, E3 +37927.810}
SPL {X  -147.202, Y  +326.099, Z    +0.000, E1   +50.843, E3 +37944.604}
SPL {X  -143.559, Y  +318.154, Z    +0.000, E1   +50.126, E3 +37960.751}
SPL {X  -132.920, Y  +299.736, Z    +0.000, E1   +44.141, E3 +38041.895}
ENDSPLINE

SPLINE
SPL {X  -143.903, Y  +318.857, Z    +0.000, E1   +34.827, E3 +38106.043}
SPL {X  -153.845, Y  +344.850, Z    +0.000, E1   +24.318, E3 +38132.138}
SPL {X  -158.184, Y  +364.762, Z    +0.000, E1   +14.458, E3 +38141.518}
SPL {X  -159.644, Y  +378.137, Z    +0.000, E1    +6.763, E3 +38144.831}
SPL {X  -159.957, Y  +385.097, Z    +0.000, E1    +2.214, E3 +38145.748}
SPL {X  -160.000, Y  +390.467, Z    +0.000, E1    -1.886, E3 +38146.188}
SPL {X  -160.000, Y  +396.882, Z    +0.000, E1    -9.361, E3 +38146.941}
SPL {X  -160.000, Y  +403.298, Z    +0.000, E1   -17.340, E3 +38148.244}
SPL {X  -160.000, Y  +414.216, Z    +0.000, E1   -29.557, E3 +38151.794}
SPL {X  -160.000, Y  +448.199, Z    +0.000, E1   -47.246, E3 +38174.286}
SPL {X  -160.000, Y  +510.996, Z    +0.000, E1   -52.996, E3 +38246.610}
SPL {X  -160.000, Y  +527.680, Z    +0.000, E1   -53.008, E3 +38273.379}
SPL {X  -160.000, Y  +543.568, Z    +0.000, E1   -52.978, E3 +38298.919}
SPL {X  -160.000, Y  +558.178, Z    +0.000, E1   -52.971, E3 +38322.379}
SPL {X  -160.000, Y  +573.149, Z    +0.000, E1   -52.983, E3 +38346.393}
SPL {X  -160.000, Y  +589.074, Z    +0.000, E1   -52.998, E3 +38371.933}
SPL {X  -160.000, Y  +605.389, Z    +0.000, E1   -52.996, E3 +38398.133}
SPL {X  -160.000, Y  +621.194, Z    +0.000, E1   -52.986, E3 +38423.533}
SPL {X  -160.000, Y  +634.261, Z    +0.000, E1   -52.926, E3 +38444.613}
SPL {X  -160.000, Y  +645.165, Z    +0.000, E1   -52.917, E3 +38462.132}
SPL {X  -160.000, Y  +655.362, Z    +0.000, E1   -52.919, E3 +38478.483}
SPL {X  -160.000, Y  +666.642, Z    +0.000, E1   -52.938, E3 +38496.558}
SPL {X  -159.882, Y  +677.646, Z    +0.000, E1   -52.897, E3 +38514.390}
SPL {X  -159.100, Y  +688.445, Z    +0.000, E1   -52.790, E3 +38532.512}
SPL {X  -157.767, Y  +698.140, Z    +0.000, E1   -52.527, E3 +38549.523}
SPL {X  -155.944, Y  +707.296, Z    +0.000, E1   -52.232, E3 +38566.081}
SPL {X  -153.388, Y  +717.020, Z    +0.000, E1   -51.781, E3 +38584.286}
SPL {X  -150.628, Y  +725.455, Z    +0.000, E1   -51.252, E3 +38600.645}
SPL {X  -147.586, Y  +733.294, Z    +0.000, E1   -50.691, E3 +38616.222}
SPL {X  -144.002, Y  +741.239, Z    +0.000, E1   -50.009, E3 +38632.398}
SPL {X  -134.968, Y  +757.427, Z    +0.000, E1   -43.006, E3 +38717.676}
ENDSPLINE

SPLINE
SPL {X  -150.251, Y  +726.498, Z    +0.000, E1   -29.147, E3 +38792.661}
SPL {X  -158.295, Y  +694.796, Z    +0.000, E1   -14.337, E3 +38810.653}
SPL {X  -159.852, Y  +678.369, Z    +0.000, E1    -4.607, E3 +38814.598}
SPL {X  -159.994, Y  +672.856, Z    +0.000, E1    -0.741, E3 +38815.185}
SPL {X  -160.000, Y  +667.974, Z    +0.000, E1    +3.384, E3 +38815.613}
SPL {X  -160.000, Y  +657.936, Z    +0.000, E1   +15.171, E3 +38817.366}
SPL {X  -160.000, Y  +643.339, Z    +0.000, E1   +31.330, E3 +38822.357}
SPL {X  -160.000, Y  +606.884, Z    +0.000, E1   +47.933, E3 +38848.213}
SPL {X  -160.000, Y  +552.863, Z    +0.000, E1   +52.205, E3 +38914.017}
SPL {X  -160.000, Y  +541.250, Z    +0.000, E1   +52.128, E3 +38933.321}
SPL {X  -160.000, Y  +532.225, Z    +0.000, E1   +52.130, E3 +38948.229}
SPL {X  -160.000, Y  +522.908, Z    +0.000, E1   +52.129, E3 +38963.633}
SPL {X  -160.000, Y  +514.018, Z    +0.000, E1   +52.121, E3 +38978.317}
SPL {X  -160.000, Y  +502.148, Z    +0.000, E1   +52.197, E3 +38997.793}
SPL {X  -160.000, Y  +488.825, Z    +0.000, E1   +51.737, E3 +39022.838}
ENDSPLINE

SPLINE
SPL {X  -160.000, Y  +489.568, Z    +0.000, E1   +48.224, E3 +39041.862}
ENDSPLINE

SPLINE
SPL {X  -160.000, Y  +479.301, Z    +0.000, E1   +49.113, E3 +39055.740}
SPL {X  -160.000, Y  +468.407, Z    +0.000, E1   +50.011, E3 +39070.067}
SPL {X  -160.000, Y  +457.258, Z    +0.000, E1   +50.929, E3 +39084.053}
SPL {X  -160.000, Y  +444.555, Z    +0.000, E1   +51.931, E3 +39099.537}
SPL {X  -160.000, Y  +432.374, Z    +0.000, E1   +52.787, E3 +39114.161}
SPL {X  -160.000, Y  +422.570, Z    +0.000, E1   +53.120, E3 +39127.919}
SPL {X  -160.000, Y  +412.343, Z    +0.000, E1   +53.116, E3 +39144.226}
SPL {X  -160.000, Y  +402.505, Z    +0.000, E1   +53.115, E3 +39159.899}
SPL {X  -160.000, Y  +391.565, Z    +0.000, E1   +53.135, E3 +39177.306}
SPL {X  -159.782, Y  +380.451, Z    +0.000, E1   +53.086, E3 +39195.268}
SPL {X  -159.005, Y  +370.988, Z    +0.000, E1   +52.949, E3 +39211.167}
SPL {X  -157.765, Y  +362.152, Z    +0.000, E1   +52.730, E3 +39226.565}
SPL {X  -156.057, Y  +353.496, Z    +0.000, E1   +52.443, E3 +39242.104}
SPL {X  -153.530, Y  +343.760, Z    +0.000, E1   +52.025, E3 +39260.157}
SPL {X  -150.540, Y  +334.599, Z    +0.000, E1   +51.451, E3 +39277.805}
SPL {X  -147.202, Y  +326.099, Z    +0.000, E1   +50.843, E3 +39294.599}
SPL {X  -143.559, Y  +318.154, Z    +0.000, E1   +50.126, E3 +39310.746}
SPL {X  -132.920, Y  +299.736, Z    +0.000, E1   +44.141, E3 +39391.891}
ENDSPLINE

SPLINE
SPL {X  -143.903, Y  +318.857, Z    +0.000, E1   +34.827, E3 +39456.038}
SPL {X  -153.845, Y  +344.850, Z    +0.000, E1   +24.318, E3 +39482.133}
SPL {X  -158.184, Y  +364.762, Z    +0.000, E1   +14.458, E3 +39491.513}
SPL {X  -159.644, Y  +378.137, Z    +0.000, E1    +6.763, E3 +39494.826}
SPL {X  -159.957, Y  +385.097, Z    +0.000, E1    +2.214, E3 +39495.743}
SPL {X  -160.000, Y  +390.467, Z    +0.000, E1    -1.886, E3 +39496.184}
SPL {X  -160.000, Y  +396.882, Z    +0.000, E1    -9.361, E3 +39496.936}
SPL {X  -160.000, Y  +403.298, Z    +0.000, E1   -17.340, E3 +39498.239}
SPL {X  -160.000, Y  +414.216, Z    +0.000, E1   -29.557, E3 +39501.789}
SPL {X  -160.000, Y  +448.199, Z    +0.000, E1   -47.246, E3 +39524.282}
SPL {X  -160.000, Y  +510.996, Z    +0.000, E1   -52.996, E3 +39596.605}
SPL {X  -160.000, Y  +527.680, Z    +0.000, E1   -53.008, E3 +39623.374}
SPL {X  -160.000, Y  +543.568, Z    +0.000, E1   -52.978, E3 +39648.914}
SPL {X  -160.000, Y  +558.178, Z    +0.000, E1   -52.971, E3 +39672.374}
SPL {X  -160.000, Y  +573.149, Z    +0.000, E1   -52.983, E3 +39696.388}
SPL {X  -160.000, Y  +589.074, Z    +0.000, E1   -52.998, E3 +39721.928}
SPL {X  -160.000, Y  +605.389, Z    +0.000, E1   -52.996, E3 +39748.129}
SPL {X  -160.000, Y  +621.194, Z    +0.000, E1   -52.986, E3 +39773.528}
SPL {X  -160.000, Y  +634.261, Z    +0.000, E1   -52.926, E3 +39794.608}
SPL {X  -160.000, Y  +645.165, Z    +0.000, E1   -52.917, E3 +39812.127}
SPL {X  -160.000, Y  +655.362, Z    +0.000, E1   -52.919, E3 +39828.478}
SPL {X  -160.000, Y  +666.642, Z    +0.000, E1   -52.938, E3 +39846.553}
SPL {X  -159.882, Y  +677.646, Z    +0.000, E1   -52.897, E3 +39864.385}
SPL {X  -159.100, Y  +688.445, Z    +0.000, E1   -52.790, E3 +39882.507}
SPL {X  -157.767, Y  +698.140, Z    +0.000, E1   -52.527, E3 +39899.518}
SPL {X  -155.944, Y  +707.296, Z    +0.000, E1   -52.232, E3 +39916.077}
SPL {X  -153.388, Y  +717.020, Z    +0.000, E1   -51.781, E3 +39934.282}
SPL {X  -150.628, Y  +725.455, Z    +0.000, E1   -51.252, E3 +39950.640}
SPL {X  -147.586, Y  +733.294, Z    +0.000, E1   -50.691, E3 +39966.217}
SPL {X  -144.002, Y  +741.239, Z    +0.000, E1   -50.009, E3 +39982.393}
SPL {X  -134.968, Y  +757.427, Z    +0.000, E1   -43.006, E3 +40067.671}
ENDSPLINE

SPLINE
SPL {X  -150.251, Y  +726.498, Z    +0.000, E1   -29.147, E3 +40142.656}
SPL {X  -158.295, Y  +694.796, Z    +0.000, E1   -14.337, E3 +40160.649}
SPL {X  -159.852, Y  +678.369, Z    +0.000, E1    -4.607, E3 +40164.593}
SPL {X  -159.994, Y  +672.856, Z    +0.000, E1    -0.741, E3 +40165.181}
SPL {X  -160.000, Y  +667.974, Z    +0.000, E1    +3.384, E3 +40165.608}
SPL {X  -160.000, Y  +657.936, Z    +0.000, E1   +15.171, E3 +40167.361}
SPL {X  -160.000, Y  +643.339, Z    +0.000, E1   +31.330, E3 +40172.353}
SPL {X  -160.000, Y  +606.884, Z    +0.000, E1   +47.933, E3 +40198.208}
SPL {X  -160.000, Y  +552.863, Z    +0.000, E1   +52.205, E3 +40264.013}
SPL {X  -160.000, Y  +541.250, Z    +0.000, E1   +52.128, E3 +40283.317}
SPL {X  -160.000, Y  +532.225, Z    +0.000, E1   +52.130, E3 +40298.224}
SPL {X  -160.000, Y  +522.908, Z    +0.000, E1   +52.129, E3 +40313.628}
SPL {X  -160.000, Y  +514.018, Z    +0.000, E1   +52.121, E3 +40328.313}
SPL {X  -160.000, Y  +502.148, Z    +0.000, E1   +52.197, E3 +40347.789}
SPL {X  -160.000, Y  +488.825, Z    +0.000, E1   +51.737, E3 +40372.833}
ENDSPLINE

SPLINE
SPL {X  -160.000, Y  +489.568, Z    +0.000, E1   +48.224, E3 +40391.858}
ENDSPLINE

SPLINE
SPL {X  -160.000, Y  +479.301, Z    +0.000, E1   +49.113, E3 +40405.736}
SPL {X  -160.000, Y  +468.407, Z    +0.000, E1   +50.011, E3 +40420.062}
SPL {X  -160.000, Y  +457.258, Z    +0.000, E1   +50.929, E3 +40434.048}
SPL {X  -160.000, Y  +444.555, Z    +0.000, E1   +51.931, E3 +40449.532}
SPL {X  -160.000, Y  +432.374, Z    +0.000, E1   +52.787, E3 +40464.156}
SPL {X  -160.000, Y  +422.570, Z    +0.000, E1   +53.120, E3 +40477.914}
SPL {X  -160.000, Y  +412.343, Z    +0.000, E1   +53.116, E3 +40494.221}
SPL {X  -160.000, Y  +402.505, Z    +0.000, E1   +53.115, E3 +40509.894}
SPL {X  -160.000, Y  +391.565, Z    +0.000, E1   +53.135, E3 +40527.301}
SPL {X  -159.782, Y  +380.451, Z    +0.000, E1   +53.086, E3 +40545.263}
SPL {X  -159.005, Y  +370.988, Z    +0.000, E1   +52.949, E3 +40561.162}
SPL {X  -157.765, Y  +362.152, Z    +0.000, E1   +52.730, E3 +40576.561}
SPL {X  -156.057, Y  +353.496, Z    +0.000, E1   +52.443, E3 +40592.099}
SPL {X  -153.530, Y  +343.760, Z    +0.000, E1   +52.025, E3 +40610.152}
SPL {X  -150.540, Y  +334.599, Z    +0.000, E1   +51.451, E3 +40627.801}
SPL {X  -147.202, Y  +326.099, Z    +0.000, E1   +50.843, E3 +40644.594}
SPL {X  -143.559, Y  +318.154, Z    +0.000, E1   +50.126, E3 +40660.741}
SPL {X  -132.920, Y  +299.736, Z    +0.000, E1   +44.141, E3 +40741.886}
ENDSPLINE

SPLINE
SPL {X  -143.903, Y  +318.857, Z    +0.000, E1   +34.827, E3 +40806.033}
SPL {X  -153.845, Y  +344.850, Z    +0.000, E1   +24.318, E3 +40832.129}
SPL {X  -158.184, Y  +364.762, Z    +0.000, E1   +14.458, E3 +40841.508}
SPL {X  -159.644, Y  +378.137, Z    +0.000, E1    +6.763, E3 +40844.822}
SPL {X  -159.957, Y  +385.097, Z    +0.000, E1    +2.214, E3 +40845.738}
SPL {X  -160.000, Y  +390.467, Z    +0.000, E1    -1.886, E3 +40846.179}
SPL {X  -160.000, Y  +396.882, Z    +0.000, E1    -9.361, E3 +40846.932}
SPL {X  -160.000, Y  +403.298, Z    +0.000, E1   -17.340, E3 +40848.234}
SPL {X  -160.000, Y  +414.216, Z    +0.000, E1   -29.557, E3 +40851.784}
SPL {X  -160.000, Y  +448.199, Z    +0.000, E1   -47.246, E3 +40874.277}
SPL {X  -160.000, Y  +510.996, Z    +0.000, E1   -52.996, E3 +40946.601}
SPL {X  -160.000, Y  +527.680, Z    +0.000, E1   -53.008, E3 +40973.369}
SPL {X  -160.000, Y  +543.568, Z    +0.000, E1   -52.978, E3 +40998.909}
SPL {X  -160.000, Y  +558.178, Z    +0.000, E1   -52.971, E3 +41022.369}
SPL {X  -160.000, Y  +573.149, Z    +0.000, E1   -52.983, E3 +41046.383}
SPL {X  -160.000, Y  +589.074, Z    +0.000, E1   -52.998, E3 +41071.923}
SPL {X  -160.000, Y  +605.389, Z    +0.000, E1   -52.996, E3 +41098.124}
SPL {X  -160.000, Y  +621.194, Z    +0.000, E1   -52.986, E3 +41123.523}
SPL {X  -160.000, Y  +634.261, Z    +0.000, E1   -52.926, E3 +41144.603}
SPL {X  -160.000, Y  +645.165, Z    +0.000, E1   -52.917, E3 +41162.122}
SPL {X  -160.000, Y  +655.362, Z    +0.000, E1   -52.919, E3 +41178.473}
SPL {X  -160.000, Y  +666.642, Z    +0.000, E1   -52.938, E3 +41196.548}
SPL {X  -159.882, Y  +677.646, Z    +0.000, E1   -52.897, E3 +41214.380}
SPL {X  -159.100, Y  +688.445, Z    +0.000, E1   -52.790, E3 +41232.502}
SPL {X  -157.767, Y  +698.140, Z    +0.000, E1   -52.527, E3 +41249.514}
SPL {X  -155.944, Y  +707.296, Z    +0.000, E1   -52.232, E3 +41266.072}
SPL {X  -153.388, Y  +717.020, Z    +0.000, E1   -51.781, E3 +41284.277}
SPL {X  -150.628, Y  +725.455, Z    +0.000, E1   -51.252, E3 +41300.635}
SPL {X  -147.586, Y  +733.294, Z    +0.000, E1   -50.691, E3 +41316.212}
SPL {X  -144.002, Y  +741.239, Z    +0.000, E1   -50.009, E3 +41332.388}
SPL {X  -134.968, Y  +757.427, Z    +0.000, E1   -43.006, E3 +41417.666}
ENDSPLINE

SPLINE
SPL {X  -150.251, Y  +726.498, Z    +0.000, E1   -29.147, E3 +41492.652}
SPL {X  -158.295, Y  +694.796, Z    +0.000, E1   -14.337, E3 +41510.644}
SPL {X  -159.852, Y  +678.369, Z    +0.000, E1    -4.607, E3 +41514.588}
SPL {X  -159.994, Y  +672.856, Z    +0.000, E1    -0.741, E3 +41515.176}
SPL {X  -160.000, Y  +667.974, Z    +0.000, E1    +3.384, E3 +41515.604}
SPL {X  -160.000, Y  +657.936, Z    +0.000, E1   +15.171, E3 +41517.356}
SPL {X  -160.000, Y  +643.339, Z    +0.000, E1   +31.330, E3 +41522.348}
SPL {X  -160.000, Y  +606.884, Z    +0.000, E1   +47.933, E3 +41548.203}
SPL {X  -160.000, Y  +552.863, Z    +0.000, E1   +52.205, E3 +41614.008}
SPL {X  -160.000, Y  +541.250, Z    +0.000, E1   +52.128, E3 +41633.312}
SPL {X  -160.000, Y  +532.225, Z    +0.000, E1   +52.130, E3 +41648.219}
SPL {X  -160.000, Y  +522.908, Z    +0.000, E1   +52.129, E3 +41663.623}
SPL {X  -160.000, Y  +514.018, Z    +0.000, E1   +52.121, E3 +41678.308}
SPL {X  -160.000, Y  +502.148, Z    +0.000, E1   +52.197, E3 +41697.784}
SPL {X  -160.000, Y  +488.825, Z    +0.000, E1   +51.737, E3 +41722.829}
ENDSPLINE

SPLINE
SPL {X  -160.000, Y  +489.568, Z    +0.000, E1   +48.224, E3 +41741.853}
ENDSPLINE

SPLINE
SPL {X  -160.000, Y  +479.301, Z    +0.000, E1   +49.113, E3 +41755.731}
SPL {X  -160.000, Y  +468.407, Z    +0.000, E1   +50.011, E3 +41770.057}
SPL {X  -160.000, Y  +457.258, Z    +0.000, E1   +50.929, E3 +41784.043}
SPL {X  -160.000, Y  +444.555, Z    +0.000, E1   +51.931, E3 +41799.527}
SPL {X  -160.000, Y  +432.374, Z    +0.000, E1   +52.787, E3 +41814.151}
SPL {X  -160.000, Y  +422.570, Z    +0.000, E1   +53.120, E3 +41827.910}
SPL {X  -160.000, Y  +412.343, Z    +0.000, E1   +53.116, E3 +41844.217}
SPL {X  -160.000, Y  +402.505, Z    +0.000, E1   +53.115, E3 +41859.889}
SPL {X  -160.000, Y  +391.565, Z    +0.000, E1   +53.135, E3 +41877.296}
SPL {X  -159.782, Y  +380.451, Z    +0.000, E1   +53.086, E3 +41895.259}
SPL {X  -159.005, Y  +370.988, Z    +0.000, E1   +52.949, E3 +41911.157}
SPL {X  -157.765, Y  +362.152, Z    +0.000, E1   +52.730, E3 +41926.556}
SPL {X  -156.057, Y  +353.496, Z    +0.000, E1   +52.443, E3 +41942.095}
SPL {X  -153.530, Y  +343.760, Z    +0.000, E1   +52.025, E3 +41960.147}
SPL {X  -150.540, Y  +334.599, Z    +0.000, E1   +51.451, E3 +41977.796}
SPL {X  -147.202, Y  +326.099, Z    +0.000, E1   +50.843, E3 +41994.589}
SPL {X  -143.559, Y  +318.154, Z    +0.000, E1   +50.126, E3 +42010.737}
SPL {X  -132.920, Y  +299.736, Z    +0.000, E1   +44.141, E3 +42091.881}
ENDSPLINE

SPLINE
SPL {X  -143.903, Y  +318.857, Z    +0.000, E1   +34.827, E3 +42156.029}
SPL {X  -153.845, Y  +344.850, Z    +0.000, E1   +24.318, E3 +42182.124}
SPL {X  -158.184, Y  +364.762, Z    +0.000, E1   +14.458, E3 +42191.503}
SPL {X  -159.644, Y  +378.137, Z    +0.000, E1    +6.763, E3 +42194.817}
SPL {X  -159.957, Y  +385.097, Z    +0.000, E1    +2.214, E3 +42195.734}
SPL {X  -160.000, Y  +390.467, Z    +0.000, E1    -1.886, E3 +42196.174}
SPL {X  -160.000, Y  +396.882, Z    +0.000, E1    -9.361, E3 +42196.927}
SPL {X  -160.000, Y  +403.298, Z    +0.000, E1   -17.340, E3 +42198.230}
SPL {X  -160.000, Y  +414.216, Z    +0.000, E1   -29.557, E3 +42201.779}
SPL {X  -160.000, Y  +448.199, Z    +0.000, E1   -47.246, E3 +42224.272}
SPL {X  -160.000, Y  +510.996, Z    +0.000, E1   -52.996, E3 +42296.596}
SPL {X  -160.000, Y  +527.680, Z    +0.000, E1   -53.008, E3 +42323.365}
SPL {X  -160.000, Y  +543.568, Z    +0.000, E1   -52.978, E3 +42348.905}
SPL {X  -160.000, Y  +558.178, Z    +0.000, E1   -52.971, E3 +42372.364}
SPL {X  -160.000, Y  +573.149, Z    +0.000, E1   -52.983, E3 +42396.378}
SPL {X  -160.000, Y  +589.074, Z    +0.000, E1   -52.998, E3 +42421.919}
SPL {X  -160.000, Y  +605.389, Z    +0.000, E1   -52.996, E3 +42448.119}
SPL {X  -160.000, Y  +621.194, Z    +0.000, E1   -52.986, E3 +42473.519}
SPL {X  -160.000, Y  +634.261, Z    +0.000, E1   -52.926, E3 +42494.598}
SPL {X  -160.000, Y  +645.165, Z    +0.000, E1   -52.917, E3 +42512.117}
SPL {X  -160.000, Y  +655.362, Z    +0.000, E1   -52.919, E3 +42528.469}
SPL {X  -160.000, Y  +666.642, Z    +0.000, E1   -52.938, E3 +42546.544}
SPL {X  -159.882, Y  +677.646, Z    +0.000, E1   -52.897, E3 +42564.375}
SPL {X  -159.100, Y  +688.445, Z    +0.000, E1   -52.790, E3 +42582.498}
SPL {X  -157.767, Y  +698.140, Z    +0.000, E1   -52.527, E3 +42599.509}
SPL {X  -155.944, Y  +707.296, Z    +0.000, E1   -52.232, E3 +42616.067}
SPL {X  -153.388, Y  +717.020, Z    +0.000, E1   -51.781, E3 +42634.272}
SPL {X  -150.628, Y  +725.455, Z    +0.000, E1   -51.252, E3 +42650.630}
SPL {X  -147.586, Y  +733.294, Z    +0.000, E1   -50.691, E3 +42666.207}
SPL {X  -144.002, Y  +741.239, Z    +0.000, E1   -50.009, E3 +42682.383}
SPL {X  -134.968, Y  +757.427, Z    +0.000, E1   -43.006, E3 +42767.662}
ENDSPLINE

SPLINE
SPL {X  -150.251, Y  +726.498, Z    +0.000, E1   -29.147, E3 +42842.647}
SPL {X  -158.295, Y  +694.796, Z    +0.000, E1   -14.337, E3 +42860.639}
SPL {X  -159.852, Y  +678.369, Z    +0.000, E1    -4.607, E3 +42864.583}
SPL {X  -159.994, Y  +672.856, Z    +0.000, E1    -0.741, E3 +42865.171}
SPL {X  -160.000, Y  +667.974, Z    +0.000, E1    +3.384, E3 +42865.599}
SPL {X  -160.000, Y  +657.936, Z    +0.000, E1   +15.171, E3 +42867.351}
SPL {X  -160.000, Y  +643.339, Z    +0.000, E1   +31.330, E3 +42872.343}
SPL {X  -160.000, Y  +606.884, Z    +0.000, E1   +47.933, E3 +42898.198}
SPL {X  -160.000, Y  +552.863, Z    +0.000, E1   +52.205, E3 +42964.003}
SPL {X  -160.000, Y  +541.250, Z    +0.000, E1   +52.128, E3 +42983.307}
SPL {X  -160.000, Y  +532.225, Z    +0.000, E1   +52.130, E3 +42998.215}
SPL {X  -160.000, Y  +522.908, Z    +0.000, E1   +52.129, E3 +43013.618}
SPL {X  -160.000, Y  +514.018, Z    +0.000, E1   +52.121, E3 +43028.303}
SPL {X  -160.000, Y  +502.148, Z    +0.000, E1   +52.197, E3 +43047.779}
SPL {X  -160.000, Y  +488.825, Z    +0.000, E1   +51.737, E3 +43072.824}
ENDSPLINE

SPLINE
SPL {X  -160.000, Y  +489.568, Z    +0.000, E1   +48.224, E3 +43091.848}
ENDSPLINE

SPLINE
SPL {X  -160.000, Y  +479.301, Z    +0.000, E1   +49.113, E3 +43105.726}
SPL {X  -160.000, Y  +468.407, Z    +0.000, E1   +50.011, E3 +43120.053}
SPL {X  -160.000, Y  +457.258, Z    +0.000, E1   +50.929, E3 +43134.038}
SPL {X  -160.000, Y  +444.555, Z    +0.000, E1   +51.931, E3 +43149.522}
SPL {X  -160.000, Y  +432.374, Z    +0.000, E1   +52.787, E3 +43164.147}
SPL {X  -160.000, Y  +422.570, Z    +0.000, E1   +53.120, E3 +43177.905}
SPL {X  -160.000, Y  +412.343, Z    +0.000, E1   +53.116, E3 +43194.212}
SPL {X  -160.000, Y  +402.505, Z    +0.000, E1   +53.115, E3 +43209.885}
SPL {X  -160.000, Y  +391.565, Z    +0.000, E1   +53.135, E3 +43227.291}
SPL {X  -159.782, Y  +380.451, Z    +0.000, E1   +53.086, E3 +43245.254}
SPL {X  -159.005, Y  +370.988, Z    +0.000, E1   +52.949, E3 +43261.153}
SPL {X  -157.765, Y  +362.152, Z    +0.000, E1   +52.730, E3 +43276.551}
SPL {X  -156.057, Y  +353.496, Z    +0.000, E1   +52.443, E3 +43292.090}
SPL {X  -153.530, Y  +343.760, Z    +0.000, E1   +52.025, E3 +43310.143}
SPL {X  -150.540, Y  +334.599, Z    +0.000, E1   +51.451, E3 +43327.791}
SPL {X  -147.202, Y  +326.099, Z    +0.000, E1   +50.843, E3 +43344.585}
SPL {X  -143.559, Y  +318.154, Z    +0.000, E1   +50.126, E3 +43360.732}
SPL {X  -132.920, Y  +299.736, Z    +0.000, E1   +44.141, E3 +43441.876}
ENDSPLINE

SPLINE
SPL {X  -143.903, Y  +318.857, Z    +0.000, E1   +34.827, E3 +43506.024}
SPL {X  -153.845, Y  +344.850, Z    +0.000, E1   +24.318, E3 +43532.119}
SPL {X  -158.184, Y  +364.762, Z    +0.000, E1   +14.458, E3 +43541.499}
SPL {X  -159.644, Y  +378.137, Z    +0.000, E1    +6.763, E3 +43544.812}
SPL {X  -159.957, Y  +385.097, Z    +0.000, E1    +2.214, E3 +43545.729}
SPL {X  -160.000, Y  +390.467, Z    +0.000, E1    -1.886, E3 +43546.169}
SPL {X  -160.000, Y  +396.882, Z    +0.000, E1    -9.361, E3 +43546.922}
SPL {X  -160.000, Y  +403.298, Z    +0.000, E1   -17.340, E3 +43548.225}
SPL {X  -160.000, Y  +414.216, Z    +0.000, E1   -29.557, E3 +43551.775}
SPL {X  -160.000, Y  +448.199, Z    +0.000, E1   -47.246, E3 +43574.267}
SPL {X  -160.000, Y  +510.996, Z    +0.000, E1   -52.996, E3 +43646.591}
SPL {X  -160.000, Y  +527.680, Z    +0.000, E1   -53.008, E3 +43673.360}
SPL {X  -160.000, Y  +543.568, Z    +0.000, E1   -52.978, E3 +43698.900}
SPL {X  -160.000, Y  +558.178, Z    +0.000, E1   -52.971, E3 +43722.360}
SPL {X  -160.000, Y  +573.149, Z    +0.000, E1   -52.983, E3 +43746.374}
SPL {X  -160.000, Y  +589.074, Z    +0.000, E1   -52.998, E3 +43771.914}
SPL {X  -160.000, Y  +605.389, Z    +0.000, E1   -52.996, E3 +43798.114}
SPL {X  -160.000, Y  +621.194, Z    +0.000, E1   -52.986, E3 +43823.514}
SPL {X  -160.000, Y  +634.261, Z    +0.000, E1   -52.926, E3 +43844.594}
SPL {X  -160.000, Y  +645.165, Z    +0.000, E1   -52.917, E3 +43862.113}
SPL {X  -160.000, Y  +655.362, Z    +0.000, E1   -52.919, E3 +43878.464}
SPL {X  -160.000, Y  +666.642, Z    +0.000, E1   -52.938, E3 +43896.539}
SPL {X  -159.882, Y  +677.646, Z    +0.000, E1   -52.897, E3 +43914.371}
SPL {X  -159.100, Y  +688.445, Z    +0.000, E1   -52.790, E3 +43932.493}
SPL {X  -157.767, Y  +698.140, Z    +0.000, E1   -52.527, E3 +43949.504}
SPL {X  -155.944, Y  +707.296, Z    +0.000, E1   -52.232, E3 +43966.062}
SPL {X  -153.388, Y  +717.020, Z    +0.000, E1   -51.781, E3 +43984.267}
SPL {X  -150.628, Y  +725.455, Z    +0.000, E1   -51.252, E3 +44000.626}
SPL {X  -147.586, Y  +733.294, Z    +0.000, E1   -50.691, E3 +44016.203}
SPL {X  -144.002, Y  +741.239, Z    +0.000, E1   -50.009, E3 +44032.379}
SPL {X  -134.968, Y  +757.427, Z    +0.000, E1   -43.006, E3 +44117.657}
ENDSPLINE

SPLINE
SPL {X  -150.251, Y  +726.498, Z    +0.000, E1   -29.147, E3 +44192.642}
SPL {X  -158.295, Y  +694.796, Z    +0.000, E1   -14.337, E3 +44210.634}
SPL {X  -159.852, Y  +678.369, Z    +0.000, E1    -4.607, E3 +44214.579}
SPL {X  -159.994, Y  +672.856, Z    +0.000, E1    -0.741, E3 +44215.166}
SPL {X  -160.000, Y  +667.974, Z    +0.000, E1    +3.384, E3 +44215.594}
SPL {X  -160.000, Y  +657.936, Z    +0.000, E1   +15.171, E3 +44217.347}
SPL {X  -160.000, Y  +643.339, Z    +0.000, E1   +31.330, E3 +44222.338}
SPL {X  -160.000, Y  +606.884, Z    +0.000, E1   +47.933, E3 +44248.194}
SPL {X  -160.000, Y  +552.863, Z    +0.000, E1   +52.205, E3 +44313.998}
SPL {X  -160.000, Y  +541.250, Z    +0.000, E1   +52.128, E3 +44333.302}
SPL {X  -160.000, Y  +532.225, Z    +0.000, E1   +52.130, E3 +44348.210}
SPL {X  -160.000, Y  +522.908, Z    +0.000, E1   +52.129, E3 +44363.614}
SPL {X  -160.000, Y  +514.018, Z    +0.000, E1   +52.121, E3 +44378.299}
SPL {X  -160.000, Y  +502.148, Z    +0.000, E1   +52.197, E3 +44397.775}
SPL {X  -160.000, Y  +488.825, Z    +0.000, E1   +51.737, E3 +44422.819}
ENDSPLINE

SPLINE
SPL {X  -160.000, Y  +489.568, Z    +0.000, E1   +48.224, E3 +44441.843}
ENDSPLINE

SPLINE
SPL {X  -160.000, Y  +479.301, Z    +0.000, E1   +49.113, E3 +44455.721}
SPL {X  -160.000, Y  +468.407, Z    +0.000, E1   +50.011, E3 +44470.048}
SPL {X  -160.000, Y  +457.258, Z    +0.000, E1   +50.929, E3 +44484.034}
SPL {X  -160.000, Y  +444.555, Z    +0.000, E1   +51.931, E3 +44499.518}
SPL {X  -160.000, Y  +432.374, Z    +0.000, E1   +52.787, E3 +44514.142}
SPL {X  -160.000, Y  +422.570, Z    +0.000, E1   +53.120, E3 +44527.900}
SPL {X  -160.000, Y  +412.343, Z    +0.000, E1   +53.116, E3 +44544.207}
SPL {X  -160.000, Y  +402.505, Z    +0.000, E1   +53.115, E3 +44559.880}
SPL {X  -160.000, Y  +391.565, Z    +0.000, E1   +53.135, E3 +44577.287}
SPL {X  -159.782, Y  +380.451, Z    +0.000, E1   +53.086, E3 +44595.249}
SPL {X  -159.005, Y  +370.988, Z    +0.000, E1   +52.949, E3 +44611.148}
SPL {X  -157.765, Y  +362.152, Z    +0.000, E1   +52.730, E3 +44626.546}
SPL {X  -156.057, Y  +353.496, Z    +0.000, E1   +52.443, E3 +44642.085}
SPL {X  -153.530, Y  +343.760, Z    +0.000, E1   +52.025, E3 +44660.138}
SPL {X  -150.540, Y  +334.599, Z    +0.000, E1   +51.451, E3 +44677.786}
SPL {X  -147.202, Y  +326.099, Z    +0.000, E1   +50.843, E3 +44694.580}
SPL {X  -143.559, Y  +318.154, Z    +0.000, E1   +50.126, E3 +44710.727}
SPL {X  -132.920, Y  +299.736, Z    +0.000, E1   +44.141, E3 +44791.872}
ENDSPLINE

SPLINE
SPL {X  -143.903, Y  +318.857, Z    +0.000, E1   +34.827, E3 +44856.019}
SPL {X  -153.845, Y  +344.850, Z    +0.000, E1   +24.318, E3 +44882.114}
SPL {X  -158.184, Y  +364.762, Z    +0.000, E1   +14.458, E3 +44891.494}
SPL {X  -159.644, Y  +378.137, Z    +0.000, E1    +6.763, E3 +44894.808}
SPL {X  -159.957, Y  +385.097, Z    +0.000, E1    +2.214, E3 +44895.724}
SPL {X  -160.000, Y  +390.467, Z    +0.000, E1    -1.886, E3 +44896.165}
SPL {X  -160.000, Y  +396.882, Z    +0.000, E1    -9.361, E3 +44896.918}
SPL {X  -160.000, Y  +403.298, Z    +0.000, E1   -17.340, E3 +44898.220}
SPL {X  -160.000, Y  +414.216, Z    +0.000, E1   -29.557, E3 +44901.770}
SPL {X  -160.000, Y  +448.199, Z    +0.000, E1   -47.246, E3 +44924.263}
SPL {X  -160.000, Y  +510.996, Z    +0.000, E1   -52.996, E3 +44996.586}
SPL {X  -160.000, Y  +527.680, Z    +0.000, E1   -53.008, E3 +45023.355}
SPL {X  -160.000, Y  +543.568, Z    +0.000, E1   -52.978, E3 +45048.895}
SPL {X  -160.000, Y  +558.178, Z    +0.000, E1   -52.971, E3 +45072.355}
SPL {X  -160.000, Y  +573.149, Z    +0.000, E1   -52.983, E3 +45096.369}
SPL {X  -160.000, Y  +589.074, Z    +0.000, E1   -52.998, E3 +45121.909}
SPL {X  -160.000, Y  +605.389, Z    +0.000, E1   -52.996, E3 +45148.110}
SPL {X  -160.000, Y  +621.194, Z    +0.000, E1   -52.986, E3 +45173.509}
SPL {X  -160.000, Y  +634.261, Z    +0.000, E1   -52.926, E3 +45194.589}
SPL {X  -160.000, Y  +645.165, Z    +0.000, E1   -52.917, E3 +45212.108}
SPL {X  -160.000, Y  +655.362, Z    +0.000, E1   -52.919, E3 +45228.459}
SPL {X  -160.000, Y  +666.642, Z    +0.000, E1   -52.938, E3 +45246.534}
SPL {X  -159.882, Y  +677.646, Z    +0.000, E1   -52.897, E3 +45264.366}
SPL {X  -159.100, Y  +688.445, Z    +0.000, E1   -52.790, E3 +45282.488}
SPL {X  -157.767, Y  +698.140, Z    +0.000, E1   -52.527, E3 +45299.500}
SPL {X  -155.944, Y  +707.296, Z    +0.000, E1   -52.232, E3 +45316.058}
SPL {X  -153.388, Y  +717.020, Z    +0.000, E1   -51.781, E3 +45334.263}
SPL {X  -150.628, Y  +725.455, Z    +0.000, E1   -51.252, E3 +45350.621}
SPL {X  -147.586, Y  +733.294, Z    +0.000, E1   -50.691, E3 +45366.198}
SPL {X  -144.002, Y  +741.239, Z    +0.000, E1   -50.009, E3 +45382.374}
SPL {X  -134.968, Y  +757.427, Z    +0.000, E1   -43.006, E3 +45467.652}
ENDSPLINE

SPLINE
SPL {X  -150.251, Y  +726.498, Z    +0.000, E1   -29.147, E3 +45542.638}
SPL {X  -158.295, Y  +694.796, Z    +0.000, E1   -14.337, E3 +45560.630}
SPL {X  -159.852, Y  +678.369, Z    +0.000, E1    -4.607, E3 +45564.574}
SPL {X  -159.994, Y  +672.856, Z    +0.000, E1    -0.741, E3 +45565.162}
SPL {X  -160.000, Y  +667.974, Z    +0.000, E1    +3.384, E3 +45565.589}
SPL {X  -160.000, Y  +657.936, Z    +0.000, E1   +15.171, E3 +45567.342}
SPL {X  -160.000, Y  +643.339, Z    +0.000, E1   +31.330, E3 +45572.334}
SPL {X  -160.000, Y  +606.884, Z    +0.000, E1   +47.933, E3 +45598.189}
SPL {X  -160.000, Y  +552.863, Z    +0.000, E1   +52.205, E3 +45663.994}
SPL {X  -160.000, Y  +541.250, Z    +0.000, E1   +52.128, E3 +45683.298}
SPL {X  -160.000, Y  +532.225, Z    +0.000, E1   +52.130, E3 +45698.205}
SPL {X  -160.000, Y  +522.908, Z    +0.000, E1   +52.129, E3 +45713.609}
SPL {X  -160.000, Y  +514.018, Z    +0.000, E1   +52.121, E3 +45728.294}
SPL {X  -160.000, Y  +502.148, Z    +0.000, E1   +52.197, E3 +45747.770}
SPL {X  -160.000, Y  +488.825, Z    +0.000, E1   +51.737, E3 +45772.814}
ENDSPLINE

SPLINE
SPL {X  -160.000, Y  +489.568, Z    +0.000, E1   +48.224, E3 +45791.839}
ENDSPLINE

SPLINE
SPL {X  -160.000, Y  +479.301, Z    +0.000, E1   +49.113, E3 +45805.717}
SPL {X  -160.000, Y  +468.407, Z    +0.000, E1   +50.011, E3 +45820.043}
SPL {X  -160.000, Y  +457.258, Z    +0.000, E1   +50.929, E3 +45834.029}
SPL {X  -160.000, Y  +444.555, Z    +0.000, E1   +51.931, E3 +45849.513}
SPL {X  -160.000, Y  +432.374, Z    +0.000, E1   +52.787, E3 +45864.137}
SPL {X  -160.000, Y  +422.570, Z    +0.000, E1   +53.120, E3 +45877.895}
SPL {X  -160.000, Y  +412.343, Z    +0.000, E1   +53.116, E3 +45894.202}
SPL {X  -160.000, Y  +402.505, Z    +0.000, E1   +53.115, E3 +45909.875}
SPL {X  -160.000, Y  +391.565, Z    +0.000, E1   +53.135, E3 +45927.282}
SPL {X  -159.782, Y  +380.451, Z    +0.000, E1   +53.086, E3 +45945.244}
SPL {X  -159.005, Y  +370.988, Z    +0.000, E1   +52.949, E3 +45961.143}
SPL {X  -157.765, Y  +362.152, Z    +0.000, E1   +52.730, E3 +45976.542}
SPL {X  -156.057, Y  +353.496, Z    +0.000, E1   +52.443, E3 +45992.080}
SPL {X  -153.530, Y  +343.760, Z    +0.000, E1   +52.025, E3 +46010.133}
SPL {X  -150.540, Y  +334.599, Z    +0.000, E1   +51.451, E3 +46027.782}
SPL {X  -147.202, Y  +326.099, Z    +0.000, E1   +50.843, E3 +46044.575}
SPL {X  -143.559, Y  +318.154, Z    +0.000, E1   +50.126, E3 +46060.722}
SPL {X  -132.920, Y  +299.736, Z    +0.000, E1   +44.141, E3 +46141.867}
ENDSPLINE

SPLINE
SPL {X  -143.903, Y  +318.857, Z    +0.000, E1   +34.827, E3 +46206.015}
SPL {X  -153.845, Y  +344.850, Z    +0.000, E1   +24.318, E3 +46232.110}
SPL {X  -158.184, Y  +364.762, Z    +0.000, E1   +14.458, E3 +46241.489}
SPL {X  -159.644, Y  +378.137, Z    +0.000, E1    +6.763, E3 +46244.803}
SPL {X  -159.957, Y  +385.097, Z    +0.000, E1    +2.214, E3 +46245.719}
SPL {X  -160.000, Y  +390.467, Z    +0.000, E1    -1.886, E3 +46246.160}
SPL {X  -160.000, Y  +396.882, Z    +0.000, E1    -9.361, E3 +46246.913}
SPL {X  -160.000, Y  +403.298, Z    +0.000, E1   -17.340, E3 +46248.215}
SPL {X  -160.000, Y  +414.216, Z    +0.000, E1   -29.557, E3 +46251.765}
SPL {X  -160.000, Y  +448.199, Z    +0.000, E1   -47.246, E3 +46274.258}
SPL {X  -160.000, Y  +510.996, Z    +0.000, E1   -52.996, E3 +46346.582}
SPL {X  -160.000, Y  +527.680, Z    +0.000, E1   -53.008, E3 +46373.350}
SPL {X  -160.000, Y  +543.568, Z    +0.000, E1   -52.978, E3 +46398.890}
SPL {X  -160.000, Y  +558.178, Z    +0.000, E1   -52.971, E3 +46422.350}
SPL {X  -160.000, Y  +573.149, Z    +0.000, E1   -52.983, E3 +46446.364}
SPL {X  -160.000, Y  +589.074, Z    +0.000, E1   -52.998, E3 +46471.904}
SPL {X  -160.000, Y  +605.389, Z    +0.000, E1   -52.996, E3 +46498.105}
SPL {X  -160.000, Y  +621.194, Z    +0.000, E1   -52.986, E3 +46523.504}
SPL {X  -160.000, Y  +634.261, Z    +0.000, E1   -52.926, E3 +46544.584}
SPL {X  -160.000, Y  +645.165, Z    +0.000, E1   -52.917, E3 +46562.103}
SPL {X  -160.000, Y  +655.362, Z    +0.000, E1   -52.919, E3 +46578.454}
SPL {X  -160.000, Y  +666.642, Z    +0.000, E1   -52.938, E3 +46596.529}
SPL {X  -159.882, Y  +677.646, Z    +0.000, E1   -52.897, E3 +46614.361}
SPL {X  -159.100, Y  +688.445, Z    +0.000, E1   -52.790, E3 +46632.483}
SPL {X  -157.767, Y  +698.140, Z    +0.000, E1   -52.527, E3 +46649.495}
SPL {X  -155.944, Y  +707.296, Z    +0.000, E1   -52.232, E3 +46666.053}
SPL {X  -153.388, Y  +717.020, Z    +0.000, E1   -51.781, E3 +46684.258}
SPL {X  -150.628, Y  +725.455, Z    +0.000, E1   -51.252, E3 +46700.616}
SPL {X  -147.586, Y  +733.294, Z    +0.000, E1   -50.691, E3 +46716.193}
SPL {X  -144.002, Y  +741.239, Z    +0.000, E1   -50.009, E3 +46732.369}
SPL {X  -134.968, Y  +757.427, Z    +0.000, E1   -43.006, E3 +46817.647}
ENDSPLINE

SPLINE
SPL {X  -150.251, Y  +726.498, Z    +0.000, E1   -29.147, E3 +46892.633}
SPL {X  -158.295, Y  +694.796, Z    +0.000, E1   -14.337, E3 +46910.625}
SPL {X  -159.852, Y  +678.369, Z    +0.000, E1    -4.607, E3 +46914.569}
SPL {X  -159.994, Y  +672.856, Z    +0.000, E1    -0.741, E3 +46915.157}
SPL {X  -160.000, Y  +667.974, Z    +0.000, E1    +3.384, E3 +46915.585}
SPL {X  -160.000, Y  +657.936, Z    +0.000, E1   +15.171, E3 +46917.337}
SPL {X  -160.000, Y  +643.339, Z    +0.000, E1   +31.330, E3 +46922.329}
SPL {X  -160.000, Y  +606.884, Z    +0.000, E1   +47.933, E3 +46948.184}
SPL {X  -160.000, Y  +552.863, Z    +0.000, E1   +52.205, E3 +47013.989}
SPL {X  -160.000, Y  +541.250, Z    +0.000, E1   +52.128, E3 +47033.293}
SPL {X  -160.000, Y  +532.225, Z    +0.000, E1   +52.130, E3 +47048.200}
SPL {X  -160.000, Y  +522.908, Z    +0.000, E1   +52.129, E3 +47063.604}
SPL {X  -160.000, Y  +514.018, Z    +0.000, E1   +52.121, E3 +47078.289}
SPL {X  -160.000, Y  +502.148, Z    +0.000, E1   +52.197, E3 +47097.765}
SPL {X  -160.000, Y  +488.825, Z    +0.000, E1   +51.737, E3 +47122.810}
ENDSPLINE

SPLINE
SPL {X  -160.000, Y  +489.568, Z    +0.000, E1   +48.224, E3 +47141.834}
ENDSPLINE

SPLINE
SPL {X  -160.000, Y  +479.301, Z    +0.000, E1   +49.113, E3 +47155.712}
SPL {X  -160.000, Y  +468.407, Z    +0.000, E1   +50.011, E3 +47170.038}
SPL {X  -160.000, Y  +457.258, Z    +0.000, E1   +50.929, E3 +47184.024}
SPL {X  -160.000, Y  +444.555, Z    +0.000, E1   +51.931, E3 +47199.508}
SPL {X  -160.000, Y  +432.374, Z    +0.000, E1   +52.787, E3 +47214.133}
SPL {X  -160.000, Y  +422.570, Z    +0.000, E1   +53.120, E3 +47227.891}
SPL {X  -160.000, Y  +412.343, Z    +0.000, E1   +53.116, E3 +47244.198}
SPL {X  -160.000, Y  +402.505, Z    +0.000, E1   +53.115, E3 +47259.870}
SPL {X  -160.000, Y  +391.565, Z    +0.000, E1   +53.135, E3 +47277.277}
SPL {X  -159.782, Y  +380.451, Z    +0.000, E1   +53.086, E3 +47295.240}
SPL {X  -159.005, Y  +370.988, Z    +0.000, E1   +52.949, E3 +47311.139}
SPL {X  -157.765, Y  +362.152, Z    +0.000, E1   +52.730, E3 +47326.537}
SPL {X  -156.057, Y  +353.496, Z    +0.000, E1   +52.443, E3 +47342.076}
SPL {X  -153.530, Y  +343.760, Z    +0.000, E1   +52.025, E3 +47360.128}
SPL {X  -150.540, Y  +334.599, Z    +0.000, E1   +51.451, E3 +47377.777}
SPL {X  -147.202, Y  +326.099, Z    +0.000, E1   +50.843, E3 +47394.570}
SPL {X  -143.559, Y  +318.154, Z    +0.000, E1   +50.126, E3 +47410.718}
SPL {X  -132.920, Y  +299.736, Z    +0.000, E1   +44.141, E3 +47491.862}
ENDSPLINE

SPLINE
SPL {X  -143.903, Y  +318.857, Z    +0.000, E1   +34.827, E3 +47556.010}
SPL {X  -153.845, Y  +344.850, Z    +0.000, E1   +24.318, E3 +47582.105}
SPL {X  -158.184, Y  +364.762, Z    +0.000, E1   +14.458, E3 +47591.484}
SPL {X  -159.644, Y  +378.137, Z    +0.000, E1    +6.763, E3 +47594.798}
SPL {X  -159.957, Y  +385.097, Z    +0.000, E1    +2.214, E3 +47595.715}
SPL {X  -160.000, Y  +390.467, Z    +0.000, E1    -1.886, E3 +47596.155}
SPL {X  -160.000, Y  +396.882, Z    +0.000, E1    -9.361, E3 +47596.908}
SPL {X  -160.000, Y  +403.298, Z    +0.000, E1   -17.340, E3 +47598.211}
SPL {X  -160.000, Y  +414.216, Z    +0.000, E1   -29.557, E3 +47601.760}
SPL {X  -160.000, Y  +448.199, Z    +0.000, E1   -47.246, E3 +47624.253}
SPL {X  -160.000, Y  +510.996, Z    +0.000, E1   -52.996, E3 +47696.577}
SPL {X  -160.000, Y  +527.680, Z    +0.000, E1   -53.008, E3 +47723.346}
SPL {X  -160.000, Y  +543.568, Z    +0.000, E1   -52.978, E3 +47748.886}
SPL {X  -160.000, Y  +558.178, Z    +0.000, E1   -52.971, E3 +47772.345}
SPL {X  -160.000, Y  +573.149, Z    +0.000, E1   -52.983, E3 +47796.359}
SPL {X  -160.000, Y  +589.074, Z    +0.000, E1   -52.998, E3 +47821.900}
SPL {X  -160.000, Y  +605.389, Z    +0.000, E1   -52.996, E3 +47848.100}
SPL {X  -160.000, Y  +621.194, Z    +0.000, E1   -52.986, E3 +47873.500}
SPL {X  -160.000, Y  +634.261, Z    +0.000, E1   -52.926, E3 +47894.579}
SPL {X  -160.000, Y  +645.165, Z    +0.000, E1   -52.917, E3 +47912.099}
SPL {X  -160.000, Y  +655.362, Z    +0.000, E1   -52.919, E3 +47928.450}
SPL {X  -160.000, Y  +666.642, Z    +0.000, E1   -52.938, E3 +47946.525}
SPL {X  -159.882, Y  +677.646, Z    +0.000, E1   -52.897, E3 +47964.356}
SPL {X  -159.100, Y  +688.445, Z    +0.000, E1   -52.790, E3 +47982.479}
SPL {X  -157.767, Y  +698.140, Z    +0.000, E1   -52.527, E3 +47999.490}
SPL {X  -155.944, Y  +707.296, Z    +0.000, E1   -52.232, E3 +48016.048}
SPL {X  -153.388, Y  +717.020, Z    +0.000, E1   -51.781, E3 +48034.253}
SPL {X  -150.628, Y  +725.455, Z    +0.000, E1   -51.252, E3 +48050.611}
SPL {X  -147.586, Y  +733.294, Z    +0.000, E1   -50.691, E3 +48066.188}
SPL {X  -144.002, Y  +741.239, Z    +0.000, E1   -50.009, E3 +48082.364}
SPL {X  -134.968, Y  +757.427, Z    +0.000, E1   -43.006, E3 +48167.643}
ENDSPLINE

SPLINE
SPL {X  -150.251, Y  +726.498, Z    +0.000, E1   -29.147, E3 +48242.628}
SPL {X  -158.295, Y  +694.796, Z    +0.000, E1   -14.337, E3 +48260.620}
SPL {X  -159.852, Y  +678.369, Z    +0.000, E1    -4.607, E3 +48264.564}
SPL {X  -159.994, Y  +672.856, Z    +0.000, E1    -0.741, E3 +48265.152}
SPL {X  -160.000, Y  +667.974, Z    +0.000, E1    +3.384, E3 +48265.580}
SPL {X  -160.000, Y  +657.936, Z    +0.000, E1   +15.171, E3 +48267.332}
SPL {X  -160.000, Y  +643.339, Z    +0.000, E1   +31.330, E3 +48272.324}
SPL {X  -160.000, Y  +606.884, Z    +0.000, E1   +47.933, E3 +48298.179}
SPL {X  -160.000, Y  +552.863, Z    +0.000, E1   +52.205, E3 +48363.984}
SPL {X  -160.000, Y  +541.250, Z    +0.000, E1   +52.128, E3 +48383.288}
SPL {X  -160.000, Y  +532.225, Z    +0.000, E1   +52.130, E3 +48398.196}
SPL {X  -160.000, Y  +522.908, Z    +0.000, E1   +52.129, E3 +48413.600}
SPL {X  -160.000, Y  +514.018, Z    +0.000, E1   +52.121, E3 +48428.284}
SPL {X  -160.000, Y  +502.148, Z    +0.000, E1   +52.197, E3 +48447.760}
SPL {X  -160.000, Y  +488.825, Z    +0.000, E1   +51.737, E3 +48472.805}
ENDSPLINE

SPLINE
SPL {X  -160.000, Y  +489.568, Z    +0.000, E1   +48.224, E3 +48491.829}
ENDSPLINE

SPLINE
SPL {X  -160.000, Y  +479.301, Z    +0.000, E1   +49.113, E3 +48505.707}
SPL {X  -160.000, Y  +468.407, Z    +0.000, E1   +50.011, E3 +48520.034}
SPL {X  -160.000, Y  +457.258, Z    +0.000, E1   +50.929, E3 +48534.019}
SPL {X  -160.000, Y  +444.555, Z    +0.000, E1   +51.931, E3 +48549.503}
SPL {X  -160.000, Y  +432.374, Z    +0.000, E1   +52.787, E3 +48564.128}
SPL {X  -160.000, Y  +422.570, Z    +0.000, E1   +53.120, E3 +48577.886}
SPL {X  -160.000, Y  +412.343, Z    +0.000, E1   +53.116, E3 +48594.193}
SPL {X  -160.000, Y  +402.505, Z    +0.000, E1   +53.115, E3 +48609.866}
SPL {X  -160.000, Y  +391.565, Z    +0.000, E1   +53.135, E3 +48627.273}
SPL {X  -159.782, Y  +380.451, Z    +0.000, E1   +53.086, E3 +48645.235}
SPL {X  -159.005, Y  +370.988, Z    +0.000, E1   +52.949, E3 +48661.134}
SPL {X  -157.765, Y  +362.152, Z    +0.000, E1   +52.730, E3 +48676.532}
SPL {X  -156.057, Y  +353.496, Z    +0.000, E1   +52.443, E3 +48692.071}
SPL {X  -153.530, Y  +343.760, Z    +0.000, E1   +52.025, E3 +48710.124}
SPL {X  -150.540, Y  +334.599, Z    +0.000, E1   +51.451, E3 +48727.772}
SPL {X  -147.202, Y  +326.099, Z    +0.000, E1   +50.843, E3 +48744.566}
SPL {X  -143.559, Y  +318.154, Z    +0.000, E1   +50.126, E3 +48760.713}
SPL {X  -132.920, Y  +299.736, Z    +0.000, E1   +44.141, E3 +48841.857}
ENDSPLINE

SPLINE
SPL {X  -143.903, Y  +318.857, Z    +0.000, E1   +34.827, E3 +48906.005}
SPL {X  -153.845, Y  +344.850, Z    +0.000, E1   +24.318, E3 +48932.100}
SPL {X  -158.184, Y  +364.762, Z    +0.000, E1   +14.458, E3 +48941.480}
SPL {X  -159.644, Y  +378.137, Z    +0.000, E1    +6.763, E3 +48944.793}
SPL {X  -159.957, Y  +385.097, Z    +0.000, E1    +2.214, E3 +48945.710}
SPL {X  -160.000, Y  +390.467, Z    +0.000, E1    -1.886, E3 +48946.151}
SPL {X  -160.000, Y  +396.882, Z    +0.000, E1    -9.361, E3 +48946.903}
SPL {X  -160.000, Y  +403.298, Z    +0.000, E1   -17.340, E3 +48948.206}
SPL {X  -160.000, Y  +414.216, Z    +0.000, E1   -29.557, E3 +48951.756}
SPL {X  -160.000, Y  +448.199, Z    +0.000, E1   -47.246, E3 +48974.248}
SPL {X  -160.000, Y  +510.996, Z    +0.000, E1   -52.996, E3 +49046.572}
SPL {X  -160.000, Y  +527.680, Z    +0.000, E1   -53.008, E3 +49073.341}
SPL {X  -160.000, Y  +543.568, Z    +0.000, E1   -52.978, E3 +49098.881}
SPL {X  -160.000, Y  +558.178, Z    +0.000, E1   -52.971, E3 +49122.341}
SPL {X  -160.000, Y  +573.149, Z    +0.000, E1   -52.983, E3 +49146.355}
SPL {X  -160.000, Y  +589.074, Z    +0.000, E1   -52.998, E3 +49171.895}
SPL {X  -160.000, Y  +605.389, Z    +0.000, E1   -52.996, E3 +49198.095}
SPL {X  -160.000, Y  +621.194, Z    +0.000, E1   -52.986, E3 +49223.495}
SPL {X  -160.000, Y  +634.261, Z    +0.000, E1   -52.926, E3 +49244.575}
SPL {X  -160.000, Y  +645.165, Z    +0.000, E1   -52.917, E3 +49262.094}
SPL {X  -160.000, Y  +655.362, Z    +0.000, E1   -52.919, E3 +49278.445}
SPL {X  -160.000, Y  +666.642, Z    +0.000, E1   -52.938, E3 +49296.520}
SPL {X  -159.882, Y  +677.646, Z    +0.000, E1   -52.897, E3 +49314.352}
SPL {X  -159.100, Y  +688.445, Z    +0.000, E1   -52.790, E3 +49332.474}
SPL {X  -157.767, Y  +698.140, Z    +0.000, E1   -52.527, E3 +49349.485}
SPL {X  -155.944, Y  +707.296, Z    +0.000, E1   -52.232, E3 +49366.043}
SPL {X  -153.388, Y  +717.020, Z    +0.000, E1   -51.781, E3 +49384.248}
SPL {X  -150.628, Y  +725.455, Z    +0.000, E1   -51.252, E3 +49400.607}
SPL {X  -147.586, Y  +733.294, Z    +0.000, E1   -50.691, E3 +49416.184}
SPL {X  -144.002, Y  +741.239, Z    +0.000, E1   -50.009, E3 +49432.360}
SPL {X  -134.968, Y  +757.427, Z    +0.000, E1   -43.006, E3 +49517.638}
ENDSPLINE

SPLINE
SPL {X  -150.251, Y  +726.498, Z    +0.000, E1   -29.147, E3 +49592.623}
SPL {X  -158.295, Y  +694.796, Z    +0.000, E1   -14.337, E3 +49610.615}
SPL {X  -159.852, Y  +678.369, Z    +0.000, E1    -4.607, E3 +49614.560}
SPL {X  -159.994, Y  +672.856, Z    +0.000, E1    -0.741, E3 +49615.147}
SPL {X  -160.000, Y  +667.974, Z    +0.000, E1    +3.384, E3 +49615.575}
SPL {X  -160.000, Y  +657.936, Z    +0.000, E1   +15.171, E3 +49617.328}
SPL {X  -160.000, Y  +643.339, Z    +0.000, E1   +31.330, E3 +49622.319}
SPL {X  -160.000, Y  +606.884, Z    +0.000, E1   +47.933, E3 +49648.175}
SPL {X  -160.000, Y  +552.863, Z    +0.000, E1   +52.205, E3 +49713.979}
SPL {X  -160.000, Y  +541.250, Z    +0.000, E1   +52.128, E3 +49733.283}
SPL {X  -160.000, Y  +532.225, Z    +0.000, E1   +52.130, E3 +49748.191}
SPL {X  -160.000, Y  +522.908, Z    +0.000, E1   +52.129, E3 +49763.595}
SPL {X  -160.000, Y  +514.018, Z    +0.000, E1   +52.121, E3 +49778.280}
SPL {X  -160.000, Y  +502.148, Z    +0.000, E1   +52.197, E3 +49797.756}
SPL {X  -160.000, Y  +488.825, Z    +0.000, E1   +51.737, E3 +49822.800}
ENDSPLINE

SPLINE
SPL {X  -160.000, Y  +489.568, Z    +0.000, E1   +48.224, E3 +49841.824}
ENDSPLINE

SPLINE
SPL {X  -160.000, Y  +479.301, Z    +0.000, E1   +49.113, E3 +49855.702}
SPL {X  -160.000, Y  +468.407, Z    +0.000, E1   +50.011, E3 +49870.029}
SPL {X  -160.000, Y  +457.258, Z    +0.000, E1   +50.929, E3 +49884.015}
SPL {X  -160.000, Y  +444.555, Z    +0.000, E1   +51.931, E3 +49899.499}
SPL {X  -160.000, Y  +432.374, Z    +0.000, E1   +52.787, E3 +49914.123}
SPL {X  -160.000, Y  +422.570, Z    +0.000, E1   +53.120, E3 +49927.881}
SPL {X  -160.000, Y  +412.343, Z    +0.000, E1   +53.116, E3 +49944.188}
SPL {X  -160.000, Y  +402.505, Z    +0.000, E1   +53.115, E3 +49959.861}
SPL {X  -160.000, Y  +391.565, Z    +0.000, E1   +53.135, E3 +49977.268}
SPL {X  -159.782, Y  +380.451, Z    +0.000, E1   +53.086, E3 +49995.230}
SPL {X  -159.005, Y  +370.988, Z    +0.000, E1   +52.949, E3 +50011.129}
SPL {X  -157.765, Y  +362.152, Z    +0.000, E1   +52.730, E3 +50026.527}
SPL {X  -156.057, Y  +353.496, Z    +0.000, E1   +52.443, E3 +50042.066}
SPL {X  -153.530, Y  +343.760, Z    +0.000, E1   +52.025, E3 +50060.119}
SPL {X  -150.540, Y  +334.599, Z    +0.000, E1   +51.451, E3 +50077.768}
SPL {X  -147.202, Y  +326.099, Z    +0.000, E1   +50.843, E3 +50094.561}
SPL {X  -143.559, Y  +318.154, Z    +0.000, E1   +50.126, E3 +50110.708}
SPL {X  -132.920, Y  +299.736, Z    +0.000, E1   +44.141, E3 +50191.853}
ENDSPLINE

SPLINE
SPL {X  -143.903, Y  +318.857, Z    +0.000, E1   +34.827, E3 +50256.000}
SPL {X  -153.845, Y  +344.850, Z    +0.000, E1   +24.318, E3 +50282.095}
SPL {X  -158.184, Y  +364.762, Z    +0.000, E1   +14.458, E3 +50291.475}
SPL {X  -159.644, Y  +378.137, Z    +0.000, E1    +6.763, E3 +50294.789}
SPL {X  -159.957, Y  +385.097, Z    +0.000, E1    +2.214, E3 +50295.705}
SPL {X  -160.000, Y  +390.467, Z    +0.000, E1    -1.886, E3 +50296.146}
SPL {X  -160.000, Y  +396.882, Z    +0.000, E1    -9.361, E3 +50296.899}
SPL {X  -160.000, Y  +403.298, Z    +0.000, E1   -17.340, E3 +50298.201}
SPL {X  -160.000, Y  +414.216, Z    +0.000, E1   -29.557, E3 +50301.751}
SPL {X  -160.000, Y  +448.199, Z    +0.000, E1   -47.246, E3 +50324.244}
SPL {X  -160.000, Y  +510.996, Z    +0.000, E1   -52.996, E3 +50396.567}
SPL {X  -160.000, Y  +527.680, Z    +0.000, E1   -53.008, E3 +50423.336}
SPL {X  -160.000, Y  +543.568, Z    +0.000, E1   -52.978, E3 +50448.876}
SPL {X  -160.000, Y  +558.178, Z    +0.000, E1   -52.971, E3 +50472.336}
SPL {X  -160.000, Y  +573.149, Z    +0.000, E1   -52.983, E3 +50496.350}
SPL {X  -160.000, Y  +589.074, Z    +0.000, E1   -52.998, E3 +50521.890}
SPL {X  -160.000, Y  +605.389, Z    +0.000, E1   -52.996, E3 +50548.091}
SPL {X  -160.000, Y  +621.194, Z    +0.000, E1   -52.986, E3 +50573.490}
SPL {X  -160.000, Y  +634.261, Z    +0.000, E1   -52.926, E3 +50594.570}
SPL {X  -160.000, Y  +645.165, Z    +0.000, E1   -52.917, E3 +50612.089}
SPL {X  -160.000, Y  +655.362, Z    +0.000, E1   -52.919, E3 +50628.440}
SPL {X  -160.000, Y  +666.642, Z    +0.000, E1   -52.938, E3 +50646.515}
SPL {X  -159.882, Y  +677.646, Z    +0.000, E1   -52.897, E3 +50664.347}
SPL {X  -159.100, Y  +688.445, Z    +0.000, E1   -52.790, E3 +50682.469}
SPL {X  -157.767, Y  +698.140, Z    +0.000, E1   -52.527, E3 +50699.481}
SPL {X  -155.944, Y  +707.296, Z    +0.000, E1   -52.232, E3 +50716.039}
SPL {X  -153.388, Y  +717.020, Z    +0.000, E1   -51.781, E3 +50734.244}
SPL {X  -150.628, Y  +725.455, Z    +0.000, E1   -51.252, E3 +50750.602}
SPL {X  -147.586, Y  +733.294, Z    +0.000, E1   -50.691, E3 +50766.179}
SPL {X  -144.002, Y  +741.239, Z    +0.000, E1   -50.009, E3 +50782.355}
SPL {X  -134.968, Y  +757.427, Z    +0.000, E1   -43.006, E3 +50867.633}
ENDSPLINE

SPLINE
SPL {X  -150.251, Y  +726.498, Z    +0.000, E1   -29.147, E3 +50942.619}
SPL {X  -158.295, Y  +694.796, Z    +0.000, E1   -14.337, E3 +50960.611}
SPL {X  -159.852, Y  +678.369, Z    +0.000, E1    -4.607, E3 +50964.555}
SPL {X  -159.994, Y  +672.856, Z    +0.000, E1    -0.741, E3 +50965.143}
SPL {X  -160.000, Y  +667.974, Z    +0.000, E1    +3.384, E3 +50965.570}
SPL {X  -160.000, Y  +657.936, Z    +0.000, E1   +15.171, E3 +50967.323}
SPL {X  -160.000, Y  +643.339, Z    +0.000, E1   +31.330, E3 +50972.315}
SPL {X  -160.000, Y  +606.884, Z    +0.000, E1   +47.933, E3 +50998.170}
SPL {X  -160.000, Y  +552.863, Z    +0.000, E1   +52.205, E3 +51063.975}
SPL {X  -160.000, Y  +541.250, Z    +0.000, E1   +52.128, E3 +51083.279}
SPL {X  -160.000, Y  +532.225, Z    +0.000, E1   +52.130, E3 +51098.186}
SPL {X  -160.000, Y  +522.908, Z    +0.000, E1   +52.129, E3 +51113.590}
SPL {X  -160.000, Y  +514.018, Z    +0.000, E1   +52.121, E3 +51128.275}
SPL {X  -160.000, Y  +502.148, Z    +0.000, E1   +52.197, E3 +51147.751}
SPL {X  -160.000, Y  +488.825, Z    +0.000, E1   +51.737, E3 +51172.796}
ENDSPLINE

SPLINE
SPL {X  -160.000, Y  +489.568, Z    +0.000, E1   +48.224, E3 +51191.820}
ENDSPLINE

SPLINE
SPL {X  -160.000, Y  +479.301, Z    +0.000, E1   +49.113, E3 +51205.698}
SPL {X  -160.000, Y  +468.407, Z    +0.000, E1   +50.011, E3 +51220.024}
SPL {X  -160.000, Y  +457.258, Z    +0.000, E1   +50.929, E3 +51234.010}
SPL {X  -160.000, Y  +444.555, Z    +0.000, E1   +51.931, E3 +51249.494}
SPL {X  -160.000, Y  +432.374, Z    +0.000, E1   +52.787, E3 +51264.118}
SPL {X  -160.000, Y  +422.570, Z    +0.000, E1   +53.120, E3 +51277.876}
SPL {X  -160.000, Y  +412.343, Z    +0.000, E1   +53.116, E3 +51294.183}
SPL {X  -160.000, Y  +402.505, Z    +0.000, E1   +53.115, E3 +51309.856}
SPL {X  -160.000, Y  +391.565, Z    +0.000, E1   +53.135, E3 +51327.263}
SPL {X  -159.782, Y  +380.451, Z    +0.000, E1   +53.086, E3 +51345.225}
SPL {X  -159.005, Y  +370.988, Z    +0.000, E1   +52.949, E3 +51361.124}
SPL {X  -157.765, Y  +362.152, Z    +0.000, E1   +52.730, E3 +51376.523}
SPL {X  -156.057, Y  +353.496, Z    +0.000, E1   +52.443, E3 +51392.061}
SPL {X  -153.530, Y  +343.760, Z    +0.000, E1   +52.025, E3 +51410.114}
SPL {X  -150.540, Y  +334.599, Z    +0.000, E1   +51.451, E3 +51427.763}
SPL {X  -147.202, Y  +326.099, Z    +0.000, E1   +50.843, E3 +51444.556}
SPL {X  -143.559, Y  +318.154, Z    +0.000, E1   +50.126, E3 +51460.703}
SPL {X  -132.920, Y  +299.736, Z    +0.000, E1   +44.141, E3 +51541.848}
ENDSPLINE

SPLINE
SPL {X  -143.903, Y  +318.857, Z    +0.000, E1   +34.827, E3 +51605.996}
SPL {X  -153.845, Y  +344.850, Z    +0.000, E1   +24.318, E3 +51632.091}
SPL {X  -158.184, Y  +364.762, Z    +0.000, E1   +14.458, E3 +51641.470}
SPL {X  -159.644, Y  +378.137, Z    +0.000, E1    +6.763, E3 +51644.784}
SPL {X  -159.957, Y  +385.097, Z    +0.000, E1    +2.214, E3 +51645.700}
SPL {X  -160.000, Y  +390.467, Z    +0.000, E1    -1.886, E3 +51646.141}
SPL {X  -160.000, Y  +396.882, Z    +0.000, E1    -9.361, E3 +51646.894}
SPL {X  -160.000, Y  +403.298, Z    +0.000, E1   -17.340, E3 +51648.197}
SPL {X  -160.000, Y  +414.216, Z    +0.000, E1   -29.557, E3 +51651.746}
SPL {X  -160.000, Y  +448.199, Z    +0.000, E1   -47.246, E3 +51674.239}
SPL {X  -160.000, Y  +510.996, Z    +0.000, E1   -52.996, E3 +51746.563}
SPL {X  -160.000, Y  +527.680, Z    +0.000, E1   -53.008, E3 +51773.331}
SPL {X  -160.000, Y  +543.568, Z    +0.000, E1   -52.978, E3 +51798.871}
SPL {X  -160.000, Y  +558.178, Z    +0.000, E1   -52.971, E3 +51822.331}
SPL {X  -160.000, Y  +573.149, Z    +0.000, E1   -52.983, E3 +51846.345}
SPL {X  -160.000, Y  +589.074, Z    +0.000, E1   -52.998, E3 +51871.885}
SPL {X  -160.000, Y  +605.389, Z    +0.000, E1   -52.996, E3 +51898.086}
SPL {X  -160.000, Y  +621.194, Z    +0.000, E1   -52.986, E3 +51923.485}
SPL {X  -160.000, Y  +634.261, Z    +0.000, E1   -52.926, E3 +51944.565}
SPL {X  -160.000, Y  +645.165, Z    +0.000, E1   -52.917, E3 +51962.084}
SPL {X  -160.000, Y  +655.362, Z    +0.000, E1   -52.919, E3 +51978.435}
SPL {X  -160.000, Y  +666.642, Z    +0.000, E1   -52.938, E3 +51996.511}
SPL {X  -159.882, Y  +677.646, Z    +0.000, E1   -52.897, E3 +52014.342}
SPL {X  -159.100, Y  +688.445, Z    +0.000, E1   -52.790, E3 +52032.464}
SPL {X  -157.767, Y  +698.140, Z    +0.000, E1   -52.527, E3 +52049.476}
SPL {X  -155.944, Y  +707.296, Z    +0.000, E1   -52.232, E3 +52066.034}
SPL {X  -153.388, Y  +717.020, Z    +0.000, E1   -51.781, E3 +52084.239}
SPL {X  -150.628, Y  +725.455, Z    +0.000, E1   -51.252, E3 +52100.597}
SPL {X  -147.586, Y  +733.294, Z    +0.000, E1   -50.691, E3 +52116.174}
SPL {X  -144.002, Y  +741.239, Z    +0.000, E1   -50.009, E3 +52132.350}
SPL {X  -134.968, Y  +757.427, Z    +0.000, E1   -43.006, E3 +52217.628}
ENDSPLINE

SPLINE
SPL {X  -150.251, Y  +726.498, Z    +0.000, E1   -29.147, E3 +52292.614}
SPL {X  -158.295, Y  +694.796, Z    +0.000, E1   -14.337, E3 +52310.606}
SPL {X  -159.852, Y  +678.369, Z    +0.000, E1    -4.607, E3 +52314.550}
SPL {X  -159.994, Y  +672.856, Z    +0.000, E1    -0.741, E3 +52315.138}
SPL {X  -160.000, Y  +667.974, Z    +0.000, E1    +3.384, E3 +52315.566}
SPL {X  -160.000, Y  +657.936, Z    +0.000, E1   +15.171, E3 +52317.318}
SPL {X  -160.000, Y  +643.339, Z    +0.000, E1   +31.330, E3 +52322.310}
SPL {X  -160.000, Y  +606.884, Z    +0.000, E1   +47.933, E3 +52348.165}
SPL {X  -160.000, Y  +552.863, Z    +0.000, E1   +52.205, E3 +52413.970}
SPL {X  -160.000, Y  +541.250, Z    +0.000, E1   +52.128, E3 +52433.274}
SPL {X  -160.000, Y  +532.225, Z    +0.000, E1   +52.130, E3 +52448.181}
SPL {X  -160.000, Y  +522.908, Z    +0.000, E1   +52.129, E3 +52463.585}
SPL {X  -160.000, Y  +514.018, Z    +0.000, E1   +52.121, E3 +52478.270}
SPL {X  -160.000, Y  +502.148, Z    +0.000, E1   +52.197, E3 +52497.746}
SPL {X  -160.000, Y  +488.825, Z    +0.000, E1   +51.737, E3 +52522.791}
ENDSPLINE

SPLINE
SPL {X  -160.000, Y  +489.568, Z    +0.000, E1   +48.224, E3 +52541.815}
ENDSPLINE

SPLINE
SPL {X  -160.000, Y  +479.301, Z    +0.000, E1   +49.113, E3 +52555.693}
SPL {X  -160.000, Y  +468.407, Z    +0.000, E1   +50.011, E3 +52570.019}
SPL {X  -160.000, Y  +457.258, Z    +0.000, E1   +50.929, E3 +52584.005}
SPL {X  -160.000, Y  +444.555, Z    +0.000, E1   +51.931, E3 +52599.489}
SPL {X  -160.000, Y  +432.374, Z    +0.000, E1   +52.787, E3 +52614.114}
ENDSPLINE

SPLINE
SPL {X  -160.000, Y  +439.051, Z    +0.000, E1   +48.624, E3 +52628.070}
SPL {X  -160.000, Y  +429.710, Z    +0.000, E1   +48.622, E3 +52645.560}
SPL {X  -160.000, Y  +420.891, Z    +0.000, E1   +48.613, E3 +52662.085}
SPL {X  -160.000, Y  +412.565, Z    +0.000, E1   +48.611, E3 +52677.650}
SPL {X  -160.000, Y  +404.943, Z    +0.000, E1   +48.601, E3 +52691.953}
SPL {X  -160.000, Y  +395.837, Z    +0.000, E1   +48.634, E3 +52708.942}
SPL {X  -159.987, Y  +386.768, Z    +0.000, E1   +48.609, E3 +52725.946}
SPL {X  -159.620, Y  +377.782, Z    +0.000, E1   +48.569, E3 +52743.114}
SPL {X  -158.761, Y  +368.924, Z    +0.000, E1   +48.401, E3 +52760.641}
SPL {X  -157.560, Y  +360.964, Z    +0.000, E1   +48.177, E3 +52776.813}
SPL {X  -156.187, Y  +354.076, Z    +0.000, E1   +47.920, E3 +52791.146}
SPL {X  -154.507, Y  +347.236, Z    +0.000, E1   +47.623, E3 +52805.674}
SPL {X  -152.108, Y  +339.169, Z    +0.000, E1   +47.215, E3 +52823.151}
SPL {X  -149.264, Y  +331.177, Z    +0.000, E1   +46.657, E3 +52840.950}
SPL {X  -146.675, Y  +324.875, Z    +0.000, E1   +46.130, E3 +52855.303}
SPL {X  -140.793, Y  +312.792, Z    +0.000, E1   +40.077, E3 +52929.546}
ENDSPLINE

SPLINE
SPL {X  -154.674, Y  +347.860, Z    +0.000, E1   +23.016, E3 +52999.689}
SPL {X  -159.179, Y  +372.617, Z    +0.000, E1   +10.186, E3 +53012.337}
SPL {X  -159.924, Y  +383.861, Z    +0.000, E1    +3.320, E3 +53014.960}
SPL {X  -160.000, Y  +389.631, Z    +0.000, E1    -0.873, E3 +53015.676}
SPL {X  -160.000, Y  +394.628, Z    +0.000, E1    -5.657, E3 +53016.351}
SPL {X  -160.000, Y  +401.354, Z    +0.000, E1   -13.067, E3 +53017.742}
SPL {X  -160.000, Y  +413.710, Z    +0.000, E1   -25.976, E3 +53022.535}
SPL {X  -160.000, Y  +449.556, Z    +0.000, E1   -44.518, E3 +53048.577}
SPL {X  -160.000, Y  +494.814, Z    +0.000, E1   -49.280, E3 +53106.926}
SPL {X  -160.000, Y  +504.699, Z    +0.000, E1   -49.282, E3 +53125.006}
SPL {X  -160.000, Y  +515.266, Z    +0.000, E1   -49.291, E3 +53144.320}
SPL {X  -160.000, Y  +526.314, Z    +0.000, E1   -49.296, E3 +53164.549}
SPL {X  -160.000, Y  +536.842, Z    +0.000, E1   -49.263, E3 +53183.875}
SPL {X  -160.000, Y  +547.071, Z    +0.000, E1   -49.286, E3 +53202.551}
SPL {X  -160.000, Y  +558.279, Z    +0.000, E1   -49.288, E3 +53223.055}
SPL {X  -160.000, Y  +568.309, Z    +0.000, E1   -49.259, E3 +53241.451}
SPL {X  -160.000, Y  +579.695, Z    +0.000, E1   -49.320, E3 +53262.181}
SPL {X  -160.000, Y  +592.166, Z    +0.000, E1   -49.294, E3 +53285.041}
SPL {X  -160.000, Y  +603.260, Z    +0.000, E1   -49.285, E3 +53305.365}
SPL {X  -160.000, Y  +615.079, Z    +0.000, E1   -49.301, E3 +53326.977}
SPL {X  -160.000, Y  +627.012, Z    +0.000, E1   -49.289, E3 +53348.830}
SPL {X  -160.000, Y  +638.544, Z    +0.000, E1   -49.285, E3 +53369.940}
SPL {X  -160.000, Y  +649.673, Z    +0.000, E1   -49.278, E3 +53390.314}
SPL {X  -160.000, Y  +661.315, Z    +0.000, E1   -49.297, E3 +53411.584}
SPL {X  -159.993, Y  +672.984, Z    +0.000, E1   -49.282, E3 +53432.974}
SPL {X  -159.528, Y  +683.783, Z    +0.000, E1   -49.201, E3 +53453.229}
SPL {X  -158.288, Y  +694.841, Z    +0.000, E1   -49.005, E3 +53474.743}
SPL {X  -156.479, Y  +704.881, Z    +0.000, E1   -48.644, E3 +53495.056}
SPL {X  -154.000, Y  +714.904, Z    +0.000, E1   -48.243, E3 +53515.866}
SPL {X  -150.967, Y  +724.498, Z    +0.000, E1   -47.642, E3 +53536.531}
SPL {X  -147.384, Y  +733.774, Z    +0.000, E1   -47.000, E3 +53557.004}
SPL {X  -139.301, Y  +750.209, Z    +0.000, E1   -41.935, E3 +53628.185}
ENDSPLINE

SPLINE
SPL {X  -151.875, Y  +721.838, Z    +0.000, E1   -27.241, E3 +53705.355}
SPL {X  -157.803, Y  +697.921, Z    +0.000, E1   -15.861, E3 +53721.222}
SPL {X  -159.710, Y  +681.128, Z    +0.000, E1    -6.465, E3 +53726.356}
SPL {X  -159.999, Y  +671.996, Z    +0.000, E1    -0.411, E3 +53727.686}
SPL {X  -160.000, Y  +665.132, Z    +0.000, E1    +5.902, E3 +53728.496}
SPL {X  -160.000, Y  +655.952, Z    +0.000, E1   +16.601, E3 +53730.491}
SPL {X  -160.000, Y  +643.612, Z    +0.000, E1   +29.091, E3 +53735.463}
SPL {X  -160.000, Y  +606.346, Z    +0.000, E1   +46.235, E3 +53763.271}
SPL {X  -160.000, Y  +564.751, Z    +0.000, E1   +49.682, E3 +53818.442}
SPL {X  -160.000, Y  +555.844, Z    +0.000, E1   +49.673, E3 +53834.523}
SPL {X  -160.000, Y  +545.889, Z    +0.000, E1   +49.702, E3 +53852.421}
SPL {X  -160.000, Y  +535.482, Z    +0.000, E1   +49.684, E3 +53871.221}
SPL {X  -160.000, Y  +526.440, Z    +0.000, E1   +49.666, E3 +53887.554}
SPL {X  -160.000, Y  +518.889, Z    +0.000, E1   +49.624, E3 +53901.379}
ENDSPLINE

SPLINE
SPL {X  -160.000, Y  +548.948, Z    +0.000, E1   +36.551, E3 +53911.067}
ENDSPLINE

SPLINE
SPL {X  -160.000, Y  +541.880, Z    +0.000, E1   +37.562, E3 +53924.845}
SPL {X  -160.000, Y  +532.200, Z    +0.000, E1   +38.842, E3 +53943.187}
SPL {X  -160.000, Y  +523.085, Z    +0.000, E1   +39.970, E3 +53959.878}
SPL {X  -160.000, Y  +513.603, Z    +0.000, E1   +41.139, E3 +53976.462}
SPL {X  -160.000, Y  +503.235, Z    +0.000, E1   +42.462, E3 +53993.170}
SPL {X  -160.000, Y  +493.516, Z    +0.000, E1   +43.493, E3 +54009.215}
SPL {X  -160.000, Y  +483.478, Z    +0.000, E1   +44.599, E3 +54024.673}
SPL {X  -160.000, Y  +473.020, Z    +0.000, E1   +45.665, E3 +54040.502}
SPL {X  -160.000, Y  +461.024, Z    +0.000, E1   +46.836, E3 +54057.978}
SPL {X  -160.000, Y  +448.988, Z    +0.000, E1   +48.043, E3 +54074.239}
SPL {X  -160.000, Y  +439.029, Z    +0.000, E1   +48.623, E3 +54089.647}
SPL {X  -160.000, Y  +429.710, Z    +0.000, E1   +48.622, E3 +54107.094}
SPL {X  -160.000, Y  +420.891, Z    +0.000, E1   +48.613, E3 +54123.619}
SPL {X  -160.000, Y  +412.565, Z    +0.000, E1   +48.611, E3 +54139.184}
SPL {X  -160.000, Y  +404.943, Z    +0.000, E1   +48.601, E3 +54153.487}
SPL {X  -160.000, Y  +395.837, Z    +0.000, E1   +48.634, E3 +54170.476}
SPL {X  -159.987, Y  +386.768, Z    +0.000, E1   +48.609, E3 +54187.481}
SPL {X  -159.620, Y  +377.782, Z    +0.000, E1   +48.569, E3 +54204.648}
SPL {X  -158.761, Y  +368.924, Z    +0.000, E1   +48.401, E3 +54222.176}
SPL {X  -157.560, Y  +360.964, Z    +0.000, E1   +48.177, E3 +54238.347}
SPL {X  -156.187, Y  +354.076, Z    +0.000, E1   +47.920, E3 +54252.680}
SPL {X  -154.507, Y  +347.236, Z    +0.000, E1   +47.623, E3 +54267.208}
SPL {X  -152.108, Y  +339.169, Z    +0.000, E1   +47.215, E3 +54284.685}
SPL {X  -149.264, Y  +331.177, Z    +0.000, E1   +46.657, E3 +54302.484}
SPL {X  -146.675, Y  +324.875, Z    +0.000, E1   +46.130, E3 +54316.837}
SPL {X  -140.793, Y  +312.792, Z    +0.000, E1   +40.077, E3 +54391.080}
ENDSPLINE

SPLINE
SPL {X  -154.674, Y  +347.860, Z    +0.000, E1   +23.016, E3 +54461.223}
SPL {X  -159.179, Y  +372.617, Z    +0.000, E1   +10.186, E3 +54473.872}
SPL {X  -159.924, Y  +383.861, Z    +0.000, E1    +3.320, E3 +54476.494}
SPL {X  -160.000, Y  +389.631, Z    +0.000, E1    -0.873, E3 +54477.210}
SPL {X  -160.000, Y  +394.628, Z    +0.000, E1    -5.657, E3 +54477.885}
SPL {X  -160.000, Y  +401.354, Z    +0.000, E1   -13.067, E3 +54479.277}
SPL {X  -160.000, Y  +413.710, Z    +0.000, E1   -25.976, E3 +54484.069}
SPL {X  -160.000, Y  +449.556, Z    +0.000, E1   -44.518, E3 +54510.111}
SPL {X  -160.000, Y  +494.814, Z    +0.000, E1   -49.280, E3 +54568.460}
SPL {X  -160.000, Y  +504.699, Z    +0.000, E1   -49.282, E3 +54586.540}
SPL {X  -160.000, Y  +515.266, Z    +0.000, E1   -49.291, E3 +54605.854}
SPL {X  -160.000, Y  +526.314, Z    +0.000, E1   -49.296, E3 +54626.083}
SPL {X  -160.000, Y  +536.842, Z    +0.000, E1   -49.263, E3 +54645.409}
SPL {X  -160.000, Y  +547.071, Z    +0.000, E1   -49.286, E3 +54664.086}
SPL {X  -160.000, Y  +558.279, Z    +0.000, E1   -49.288, E3 +54684.590}
SPL {X  -160.000, Y  +568.309, Z    +0.000, E1   -49.259, E3 +54702.985}
SPL {X  -160.000, Y  +579.695, Z    +0.000, E1   -49.320, E3 +54723.715}
SPL {X  -160.000, Y  +592.166, Z    +0.000, E1   -49.294, E3 +54746.575}
SPL {X  -160.000, Y  +603.260, Z    +0.000, E1   -49.285, E3 +54766.900}
SPL {X  -160.000, Y  +615.079, Z    +0.000, E1   -49.301, E3 +54788.512}
SPL {X  -160.000, Y  +627.012, Z    +0.000, E1   -49.289, E3 +54810.364}
SPL {X  -160.000, Y  +638.544, Z    +0.000, E1   -49.285, E3 +54831.474}
SPL {X  -160.000, Y  +649.673, Z    +0.000, E1   -49.278, E3 +54851.848}
SPL {X  -160.000, Y  +661.315, Z    +0.000, E1   -49.297, E3 +54873.118}
SPL {X  -159.993, Y  +672.984, Z    +0.000, E1   -49.282, E3 +54894.509}
SPL {X  -159.528, Y  +683.783, Z    +0.000, E1   -49.201, E3 +54914.763}
SPL {X  -158.288, Y  +694.841, Z    +0.000, E1   -49.005, E3 +54936.277}
SPL {X  -156.479, Y  +704.881, Z    +0.000, E1   -48.644, E3 +54956.591}
SPL {X  -154.000, Y  +714.904, Z    +0.000, E1   -48.243, E3 +54977.400}
SPL {X  -150.967, Y  +724.498, Z    +0.000, E1   -47.642, E3 +54998.065}
SPL {X  -147.384, Y  +733.774, Z    +0.000, E1   -47.000, E3 +55018.538}
SPL {X  -139.301, Y  +750.209, Z    +0.000, E1   -41.935, E3 +55089.719}
ENDSPLINE

